		// If the cryostat is no longer cold or operational, return to the appropriate warm state.
		IF stat.nState = E_NOTT_CRYO_CTRL_STATE.COLD
		   AND NOT (stat.bOP OR stat.bCold) THEN
			ctrl.bEnable_WarmUp := FALSE;
		
			IF stat.bVacuumOK OR stat.bVacuum THEN
				logs.M_LogInfo('Cryostat no longer cold. State is WARM_VACUUM.');
				stat.nState := E_NOTT_CRYO_CTRL_STATE.WARM_VACUUM;
			ELSE
				ctrl.bEnable_CoolDown := FALSE;
				logs.M_LogInfo('Cryostat no longer cold and vacuum not present. State is WARM_PRESS.');
				stat.nState := E_NOTT_CRYO_CTRL_STATE.WARM_PRESS;
			END_IF
		
		// Process queued top-level commands.
		ELSIF stat.nState = E_NOTT_CRYO_CTRL_STATE.COLD
		   AND ctrl.bExecute THEN
			ctrl.bExecute     := FALSE;
			stat.nLastCommand := ctrl.nCommand;
			ctrl.nCommand     := E_NOTT_CRYO_CTRL_CMD.NONE;
		
			CASE stat.nLastCommand OF
		
				E_NOTT_CRYO_CTRL_CMD.WARM_UP:
					IF warm_up.bPermitStart THEN
						logs.M_LogInfo('Warm-up started.');
		
						ctrl.bEnable_Evac     := TRUE;
						ctrl.bEnable_WarmUp   := TRUE;
						ctrl.bEnable_CoolDown := FALSE;
		
						stat.nState := E_NOTT_CRYO_CTRL_STATE.WARMING_UP;
					ELSE
						ctrl.bEnable_WarmUp := FALSE;
						logs.M_LogInfo('WARM_UP command rejected: warmup start not permitted in COLD.');
					END_IF
		
				E_NOTT_CRYO_CTRL_CMD.COOL:
					// Already cold. Cooling command is only useful if cooldown is not active
					// and permissions allow it.
					IF cool_down.bPermitStart AND cool_down.cooler.stat.bInitialised THEN
						logs.M_LogInfo('Cooldown command accepted in COLD: maintaining cold state.');
		
						ctrl.bEnable_Evac     := TRUE;
						ctrl.bEnable_CoolDown := TRUE;
						ctrl.bEnable_WarmUp   := FALSE;
					ELSE
						logs.M_LogInfo('COOL command ignored/rejected: system is already COLD or cooldown not permitted.');
					END_IF
		
			ELSE
				logs.M_LogInfo('Command rejected: unsupported command in COLD.');
			END_CASE
		
		// After cooler startup has completed, clear cooldown if the cooler stops
		// unexpectedly. START_PTC inactivity is part of normal startup.
		ELSIF stat.nState = E_NOTT_CRYO_CTRL_STATE.COLD
		   AND ctrl.bEnable_CoolDown
		   AND ((cool_down.stat.nState = E_NOTT_CRYO_COOLDOWN_STATE.COOLING)
			OR (cool_down.stat.nState = E_NOTT_CRYO_COOLDOWN_STATE.OPERATIONAL_TEMPERATURE_ACHIEVED))
		   AND NOT cool_down.cooler.stat.bActive THEN
			ctrl.bEnable_CoolDown := FALSE;
			logs.M_LogInfo('Cooldown enable cleared in COLD: cooler inactive.');
		END_IF
		
		M_SetStatus(stat.nState);
		RETURN;
	
	/////////////////////////////////
	E_NOTT_CRYO_CTRL_STATE.WARMING_UP:
	/////////////////////////////////
	//
	// Warmup routine is active or expected to be active.
	// Permissions are handled centrally in M_SetCmdPermissions().
	// The warmup routine must not be considered complete automatically when the
	// warm targets are reached. It remains active until the operator stops it.
	//
	
	// Cooldown must remain disabled during warmup.
	ctrl.bEnable_CoolDown := FALSE;
	
	// Evacuation should remain enabled/available during warmup.
	ctrl.bEnable_Evac := TRUE;
	
	// Reject queued top-level sequence commands while warmup is active.
	// Stop warmup via ctrl.bEnable_WarmUp FALSE and permission logic.
	IF ctrl.bExecute THEN
		stat.nLastCommand := ctrl.nCommand;
		ctrl.bExecute     := FALSE;
		ctrl.nCommand     := E_NOTT_CRYO_CTRL_CMD.NONE;
	
		CASE stat.nLastCommand OF
			E_NOTT_CRYO_CTRL_CMD.WARM_UP:
				logs.M_LogInfo('WARM_UP command ignored: warmup already active.');
	
			E_NOTT_CRYO_CTRL_CMD.COOL:
				logs.M_LogInfo('COOL command rejected: warmup active.');
		ELSE
				logs.M_LogInfo('Command rejected: warmup active.');
		END_CASE
	END_IF
	
	// Operator stop accepted by command/permission.
	IF NOT ctrl.bEnable_WarmUp THEN
		ctrl.bEnable_CoolDown := FALSE;
	
		IF stat.bOP OR stat.bCold THEN
			// Warmup was interrupted while still cold.
			ctrl.bEnable_Evac   := TRUE;
			ctrl.bEnable_WarmUp := FALSE;
	
			logs.M_LogInfo('Warmup stopped while cryostat is still cold. State is COLD.');
			stat.nState := E_NOTT_CRYO_CTRL_STATE.COLD;
	
		ELSIF stat.bVacuumOK OR stat.bVacuum THEN
			ctrl.bEnable_WarmUp := FALSE;
	
			logs.M_LogInfo('Warmup stopped. State is WARM_VACUUM.');
			stat.nState := E_NOTT_CRYO_CTRL_STATE.WARM_VACUUM;
	
		ELSE
			ctrl.bEnable_Evac   := FALSE;
			ctrl.bEnable_WarmUp := FALSE;
	
			logs.M_LogInfo('Warmup stopped and vacuum not present. State is WARM_PRESS.');
			stat.nState := E_NOTT_CRYO_CTRL_STATE.WARM_PRESS;
		END_IF
	
	// Warmup routine reports inactive while the top-level warmup command is still
	// enabled. Do not auto-stop or reclassify here. This can happen during startup,
	// a scan-order transient, or a routine implementation detail. The operator stop
	// above is the normal exit path from WARMING_UP.
	ELSIF NOT warm_up.stat.bActive THEN
		ctrl.bEnable_WarmUp   := TRUE;
		ctrl.bEnable_CoolDown := FALSE;
		ctrl.bEnable_Evac     := TRUE;
		stat.nState           := E_NOTT_CRYO_CTRL_STATE.WARMING_UP;
	END_IF
	
	M_SetStatus(stat.nState);
	RETURN;
	
	
	/////////////////////////////////
	E_NOTT_CRYO_CTRL_STATE.ERROR:
	/////////////////////////////////
	//
	// Fault state.
	// Keep commands and process routines disabled.
	// Use RESET to restart state estimation through NONE.
	//
	
	// Clear pending top-level command.
	ctrl.bExecute := FALSE;
	ctrl.nCommand := E_NOTT_CRYO_CTRL_CMD.NONE;
	
	// Disable process enables.
	// Depending on the failure type, evacuation might eventually need special
	// handling, but for now keep this simple and conservative.
	ctrl.bEnable_CoolDown := FALSE;
	ctrl.bEnable_WarmUp   := FALSE;
	ctrl.bEnable_Evac     := FALSE;
	
	// Permissions are handled centrally in M_SetCmdPermissions().
	// If desired later, add explicit ERROR handling there to force all permits FALSE.
	
	IF ctrl.bReset THEN
		ctrl.bReset := FALSE;
	
		// Re-run startup/state estimation after reset.
		stat.bSystemStarted := FALSE;
		stat.bError         := FALSE;
		stat.nState         := E_NOTT_CRYO_CTRL_STATE.NONE;
	
		logs.M_LogInfo('ERROR reset requested. Restarting state estimation.');
	
		M_SetStatus(stat.nState);
	
	// auto-recovery.

	(*
	ELSIF NOT stat.bError THEN
		stat.bSystemStarted := FALSE;
		stat.nState := E_NOTT_CRYO_CTRL_STATE.NONE;
	
		logs.M_LogInfo('ERROR cleared. Restarting state estimation.');
	
		M_SetStatus(stat.nState);
	*)
	END_IF
	
	M_SetStatus(stat.nState);
	RETURN;

END_CASE
END_METHOD

METHOD M_UpdateThermalStatus
VAR_INPUT
END_VAR
VAR
	lrDetectorTempK:		LREAL := 9999.0;
	bDetectorTempValid:		BOOL := FALSE;
	bOPInputsValid:			BOOL := FALSE;
	bOPEntryCondition:		BOOL := FALSE;
	bOPExitCondition:		BOOL := FALSE;
END_VAR
VAR_INST
	tonOPEntry:	TON;
	tonOPExit:	TON;
	tonColdEntry:	TON;
	tonColdExit:	TON;
END_VAR
VAR CONSTANT
	tOPEntryConfirm:	TIME := T#10S;
	tOPExitConfirm:		TIME := T#5S;
	tColdConfirm:		TIME := T#5S;
END_VAR

// COLD means the authoritative detector vote is below the warm threshold.
// OP is estimated centrally from the authoritative detector and base-plate
// voters together with VAGC pressure. Timers and separate reset thresholds
// prevent sensor noise from flickering the operational status.

bDetectorTempValid := nott_voters.vote_detector.stat.bValid;

IF bDetectorTempValid THEN
	lrDetectorTempK := nott_voters.vote_detector.stat.lrTempK;
END_IF

IF stat.bCold THEN
	tonColdEntry(IN := FALSE, PT := tColdConfirm);
	tonColdExit(
		IN := NOT bDetectorTempValid
			OR NOT stat.bPressureValid
			OR NOT stat.bVacuum
			OR (lrDetectorTempK > cfg.lrTemp_Warm_Reset),
		PT := tColdConfirm);

	IF tonColdExit.Q THEN
		stat.bCold := FALSE;
		tonColdExit(IN := FALSE, PT := tColdConfirm);
	END_IF
ELSE
	tonColdExit(IN := FALSE, PT := tColdConfirm);
	tonColdEntry(
		IN := bDetectorTempValid
			AND stat.bPressureValid
			AND stat.bVacuum
			AND (lrDetectorTempK < cfg.lrTemp_Warm),
		PT := tColdConfirm);

	IF tonColdEntry.Q THEN
		stat.bCold := TRUE;
		tonColdEntry(IN := FALSE, PT := tColdConfirm);
	END_IF
END_IF

// All required measurements must be valid before entering OP. A sustained
// validity loss also removes OP after the exit confirmation time.
bOPInputsValid :=
	nott_voters.vote_detector.stat.bValid
	AND nott_voters.vote_base_plate.stat.bValid
	AND VAGC.stat.bValid;

bOPEntryCondition :=
	bOPInputsValid
	AND (nott_voters.vote_detector.stat.lrTempK <= cfg.lrTemp_DET_Target)
	AND (nott_voters.vote_base_plate.stat.lrTempK < cfg.lrTemp_BasePlate_OP)
	AND (VAGC.stat.lrPressure < cfg.lrPress_OP);

bOPExitCondition :=
	NOT bOPInputsValid
	OR (nott_voters.vote_detector.stat.lrTempK > cfg.lrTemp_DET_OP_Reset)
	OR (nott_voters.vote_base_plate.stat.lrTempK > cfg.lrTemp_BasePlate_OP_Reset)
	OR (VAGC.stat.lrPressure > cfg.lrPress_OP_Reset);

IF stat.bOP THEN
	tonOPEntry(IN := FALSE, PT := tOPEntryConfirm);
	tonOPExit(IN := bOPExitCondition, PT := tOPExitConfirm);

	IF tonOPExit.Q THEN
		stat.bOP := FALSE;
		tonOPExit(IN := FALSE, PT := tOPExitConfirm);
	END_IF
ELSE
	tonOPExit(IN := FALSE, PT := tOPExitConfirm);
	tonOPEntry(IN := bOPEntryCondition, PT := tOPEntryConfirm);

	IF tonOPEntry.Q THEN
		stat.bOP := TRUE;
		tonOPEntry(IN := FALSE, PT := tOPEntryConfirm);
	END_IF
END_IF
RETURN;
END_METHOD

END_FUNCTION_BLOCK

// ---- POUs/Routines/CoolDown/FB_NOTT_CRYO_COOLDOWN.TcPOU
FUNCTION_BLOCK FB_NOTT_CRYO_COOLDOWN
VAR_INPUT
	in_bEnable:		BOOL := FALSE;	// System active while in_bEnable is TRUE
	in_Cryo_Stat:	T_NOTT_CRYO_STAT;
END_VAR
VAR_OUTPUT
	out_bPermit_Evacuation_Stop:	BOOL := FALSE;
	out_bPermit_WarmUp:				BOOL := FALSE;

END_VAR

VAR_IN_OUT
	{attribute 'OPC.UA.DA' := '0'}
	nott_temps:						FB_NOTT_TEMPERATURES;
	{attribute 'OPC.UA.DA' := '0'}
	nott_heaters:					FB_NOTT_HEATERS;
	{attribute 'OPC.UA.DA' := '0'}
	nott_t_ctrls:      				FB_NOTT_TCTRLs;
	{attribute 'OPC.UA.DA' := '0'}
	nott_t_votes: 					FB_NOTT_VOTERS;
END_VAR
VAR
	
	{attribute 'TcHmiSymbol.Show'}	
	cfg:	T_NOTT_CRYO_COOLDOWN_CFG;
	{attribute 'TcHmiSymbol.Show'}
	ctrl:	T_NOTT_CRYO_COOLDOWN_CTRL;

	{attribute 'OPC.UA.DA' := '1'}
	{attribute 'OPC.UA.DA.Access' := '1'}
	{attribute 'TcHmiSymbol.Show'}
	stat:	T_NOTT_CRYO_COOLDOWN_STAT;

// Cooler	
	
	{attribute 'TcHmiSymbol.Show'}
	cooler:			FB_METIS_CRYO_CPA;
	
//
// Internals
//
	timer:	TON;
	trig:	R_TRIG;	// Start trigger
//

	{attribute 'TcHmiSymbol.Show'}
	bPermitStart:	BOOL := FALSE;
	{attribute 'TcHmiSymbol.Show'}
	bPermitStop:	BOOL := FALSE;
	
END_VAR

M_Configure();
M_ExecuteControllers();
M_SafetyCheck();
M_StateMachine( 
	nott_temps  := nott_temps,
	nott_heaters := nott_heaters,
	nott_t_ctrls := nott_t_ctrls,
	nott_t_votes := nott_t_votes
);
M_UpdateStatus();

METHOD M_Configure
VAR_INPUT
END_VAR
VAR
	refBOOL:	REFERENCE TO BOOL;
END_VAR
// IF stat.bConfigured THEN
// 
// ELSE
// 	RETURN;
// END_IF
END_METHOD

METHOD M_ExecuteControllers
VAR
	ptrSimTemp:	POINTER TO LREAL;
END_VAR


	
// Hardware-level cooling veto. This prevents a stale command or scan-order
// delay from enabling the cooler before confirmed vacuum is available.
ctrl.cor_Cooler(
    in_bEnable := ctrl.bEnable_Cooler
        AND in_Cryo_Stat.bPressureValid
        AND in_Cryo_Stat.bVacuum
        AND (
            (in_Cryo_Stat.bIsPVPRunning
             AND in_Cryo_Stat.bIsTMPRunning)
            OR in_Cryo_Stat.bOP
        ));
Cooler(
	in_bEnable:= ctrl.cor_Cooler.out_bEnable,
	in_bSimulation:= FALSE, 
	in_sName:= 'PTC Cooler', 
	in_sSN_Compressor:= 'CPA28H5W2DNCE-410730000001', 
	in_sSN_PulseTube:= 'PT810-19880200001', 
	in_nYear_Compressor:= 2023, 
	in_nYear_PulseTube:= 2023, 
	in_lrNextService_Compressor:= 20000.0, 
	in_lrNextService_PulseTube:= 40000.0, 
	in_nSlaveID:= 16, 
	in_nPeriod:= 1000);
END_METHOD

METHOD M_PermitStart_Cooldown
VAR_INPUT
	in_bPermissionStart: BOOL;
END_VAR
bPermitStart := in_bPermissionStart;
END_METHOD

METHOD M_PermitStop_Cooldown
VAR_INPUT
	in_bPermissionStop: BOOL;
END_VAR
bPermitStop := in_bPermissionStop;
END_METHOD

METHOD M_SafetyCheck
VAR_INPUT
END_VAR
VAR CONSTANT
	lrPress_ColdAlarmTrip:	LREAL := 10.0E-1;	// [mbar]
	lrPress_ColdAlarmReset:	LREAL := 8.0E-1;	// [mbar], hysteresis reset
END_VAR
// Keep pressure and pump alarm causes separate so clearing one condition
// cannot hide the other.
IF NOT in_Cryo_Stat.bCold THEN
	stat.bPressureAlarm := FALSE;
ELSIF in_Cryo_Stat.bPressureValid THEN
	IF stat.bPressureAlarm THEN
		IF in_Cryo_Stat.lrPressure_mbar < lrPress_ColdAlarmReset THEN
			stat.bPressureAlarm := FALSE;
		END_IF
	ELSIF in_Cryo_Stat.lrPressure_mbar > lrPress_ColdAlarmTrip THEN
		stat.bPressureAlarm := TRUE;
	END_IF
END_IF

// A pump loss during active cooldown trips the routine. The alarm resets only
// after both pumps recover; a new operator command is required to restart.
IF stat.bActive
    AND NOT in_Cryo_Stat.bOP
    AND (NOT in_Cryo_Stat.bIsPVPRunning
         OR NOT in_Cryo_Stat.bIsTMPRunning) THEN

    stat.bPumpAlarm := TRUE;
    ctrl.bEnable_Cooler := FALSE;
    stat.nState := E_NOTT_CRYO_COOLDOWN_STATE.STOP_COOLDOWN;
    stat.sErrorText := 'Pump stopped during cooldown.';

ELSIF (in_Cryo_Stat.bIsPVPRunning
       AND in_Cryo_Stat.bIsTMPRunning)
      OR in_Cryo_Stat.bOP THEN

    stat.bPumpAlarm := FALSE;
END_IF


stat.bAlarm := stat.bPressureAlarm OR stat.bPumpAlarm;
stat.bWarning := stat.bAlarm;
END_METHOD

METHOD M_StateMachine : BOOL
VAR_INPUT
END_VAR
VAR_IN_OUT
	{attribute 'OPC.UA.DA' := '0'}
	nott_temps:						FB_NOTT_TEMPERATURES;
	{attribute 'OPC.UA.DA' := '0'}
	nott_heaters:					FB_NOTT_HEATERS;
	{attribute 'OPC.UA.DA' := '0'}
	nott_t_ctrls:      				FB_NOTT_TCTRLs;
	{attribute 'OPC.UA.DA' := '0'}
	nott_t_votes: 					FB_NOTT_VOTERS;
END_VAR
VAR_INST
    tonStopCooldown : TON;
END_VAR
M_StateMachine := FALSE;

// The routine cannot remain in a cooling state without confirmed vacuum.
// The actuator is already vetoed in M_ExecuteControllers(); this transition
// keeps the routine state and HMI status consistent with physical safety.
IF ((stat.nState = E_NOTT_CRYO_COOLDOWN_STATE.START_PTC)
	OR (stat.nState = E_NOTT_CRYO_COOLDOWN_STATE.START_RAMPDOWN_DETECTOR)
	OR (stat.nState = E_NOTT_CRYO_COOLDOWN_STATE.COOLING)
	OR (stat.nState = E_NOTT_CRYO_COOLDOWN_STATE.OPERATIONAL_TEMPERATURE_ACHIEVED))
	AND (NOT in_Cryo_Stat.bPressureValid OR NOT in_Cryo_Stat.bVacuum) THEN
	ctrl.bEnable_Cooler := FALSE;
	stat.nState := E_NOTT_CRYO_COOLDOWN_STATE.STOP_COOLDOWN;
	stat.sStatus := 'Stopping cooldown: vacuum lost or pressure invalid.';
END_IF

CASE stat.nState OF

    E_NOTT_CRYO_COOLDOWN_STATE.NONE:
        // Nothing to do here
        stat.sStatus := 'NONE';
		stat.bActive := FALSE;
		stat.nState := E_NOTT_CRYO_COOLDOWN_STATE.OFF;

    E_NOTT_CRYO_COOLDOWN_STATE.OFF:

        ctrl.cor_Cooler.M_SetPermissions(FALSE, TRUE); // Only OFF allowed

        stat.sState  := 'OFF';
        stat.sStatus := 'OFF';

        ctrl.bEnable_Cooler := FALSE;

        out_bPermit_Evacuation_Stop := TRUE;
        out_bPermit_WarmUp          := TRUE;
		stat.bActive := FALSE;
		
        trig(CLK := in_bEnable);

        IF trig.Q
		   AND in_Cryo_Stat.bPressureValid
		   AND in_Cryo_Stat.bVacuum
		   AND in_Cryo_Stat.bIsPVPRunning
		   AND in_Cryo_Stat.bIsTMPRunning THEN
            stat.nState := E_NOTT_CRYO_COOLDOWN_STATE.START_PTC;
            stat.sStatus := 'Starting PTC...';

            out_bPermit_Evacuation_Stop := FALSE;
            out_bPermit_WarmUp          := FALSE;
			
			stat.bActive := TRUE;
		ELSIF trig.Q THEN
			stat.sStatus := 'Cooldown start rejected: vacuum/pumps not ready.';
        END_IF;


    E_NOTT_CRYO_COOLDOWN_STATE.START_PTC:
		stat.bActive := TRUE;
		ctrl.cor_Cooler.M_SetPermissions(TRUE, TRUE);

		out_bPermit_Evacuation_Stop := FALSE;
		out_bPermit_WarmUp          := FALSE;

		IF NOT in_bEnable THEN
			ctrl.bEnable_Cooler := FALSE;
			stat.nState := E_NOTT_CRYO_COOLDOWN_STATE.STOP_COOLDOWN;
			stat.sStatus := 'Cooldown cancelled while starting PTC...';
		ELSE
			ctrl.bEnable_Cooler := TRUE;

			IF cooler.stat.bSystemOn THEN
				stat.nState := E_NOTT_CRYO_COOLDOWN_STATE.START_RAMPDOWN_DETECTOR;
				stat.sStatus := 'PTC started. Starting detector ramp down...';
			END_IF
		END_IF


    E_NOTT_CRYO_COOLDOWN_STATE.START_RAMPDOWN_DETECTOR:
		ctrl.cor_Cooler.M_SetPermissions(TRUE, TRUE);
		ctrl.bEnable_Cooler := TRUE;

		IF NOT in_bEnable THEN
			ctrl.bEnable_Cooler := FALSE;
			stat.nState := E_NOTT_CRYO_COOLDOWN_STATE.STOP_COOLDOWN;
			stat.sStatus := 'Stopping cooldown...';
			RETURN;
		END_IF

        // Enable detector heaters
        nott_heaters.h_detector.M_SetEnable();
        nott_heaters.h_detector_spare.M_SetEnable();

        // Enable detector temperature control loops
        nott_t_ctrls.tc_detector.M_SetEnable();
        nott_t_ctrls.tc_detector_spare.M_SetEnable();

        // Set detector setpoints
        nott_t_ctrls.tc_detector.M_Set_SetPoint(
            m_eSetpointType    := E_METIS_CTRL_SETPOINT_SWITCH.FIXED,
            m_lrFixedSetpoint  := cfg.lrTemp_Det,
            m_lrSetpointOffset := 0.0,
            m_pSetpointTemp    := nott_temps.M_SetTemperatureSensor(0)
        );

        nott_t_ctrls.tc_detector_spare.M_Set_SetPoint(
            m_eSetpointType    := E_METIS_CTRL_SETPOINT_SWITCH.FIXED,
            m_lrFixedSetpoint  := cfg.lrTemp_Det,
            m_lrSetpointOffset := 0.0,
            m_pSetpointTemp    := nott_temps.M_SetTemperatureSensor(0)
        );

        stat.sStatus := 'Detector ramp down active...';

        stat.nState := E_NOTT_CRYO_COOLDOWN_STATE.COOLING;
		stat.bActive := TRUE;

    E_NOTT_CRYO_COOLDOWN_STATE.COOLING:
		ctrl.cor_Cooler.M_SetPermissions(TRUE, TRUE);
		ctrl.bEnable_Cooler := TRUE;

        out_bPermit_Evacuation_Stop := FALSE;
        out_bPermit_WarmUp          := FALSE;
		stat.bActive := TRUE;
        IF in_bEnable THEN

            IF in_Cryo_Stat.bOP THEN

                stat.sStatus := 'Operational temperature achieved.';
                stat.nState  := E_NOTT_CRYO_COOLDOWN_STATE.OPERATIONAL_TEMPERATURE_ACHIEVED;

            ELSE
                stat.sStatus := 'Cooling...';
            END_IF;

        ELSE
            stat.nState := E_NOTT_CRYO_COOLDOWN_STATE.STOP_COOLDOWN;
            stat.sStatus := 'Stopping cooldown...';
        END_IF;


    E_NOTT_CRYO_COOLDOWN_STATE.OPERATIONAL_TEMPERATURE_ACHIEVED:
		stat.bActive := TRUE;
		ctrl.cor_Cooler.M_SetPermissions(TRUE, TRUE);
		ctrl.bEnable_Cooler := TRUE;
        IF in_bEnable THEN
			IF NOT in_Cryo_Stat.bOP THEN
				out_bPermit_Evacuation_Stop := FALSE;
				out_bPermit_WarmUp          := FALSE;
				stat.nState := E_NOTT_CRYO_COOLDOWN_STATE.COOLING;
				stat.sStatus := 'Operational state lost. Resuming cooldown...';
			ELSE
                stat.sStatus := 'Operational temperature achieved.';

                out_bPermit_Evacuation_Stop := TRUE;
                out_bPermit_WarmUp          := FALSE;
			END_IF

        ELSE
            stat.nState := E_NOTT_CRYO_COOLDOWN_STATE.STOP_COOLDOWN;
            stat.sStatus := 'Stopping cooldown...';

            out_bPermit_Evacuation_Stop := FALSE;
            out_bPermit_WarmUp          := FALSE;
        END_IF;


    E_NOTT_CRYO_COOLDOWN_STATE.STOP_COOLDOWN:
		stat.bActive := TRUE;
		// Disable PTC
		ctrl.cor_Cooler.M_SetPermissions(FALSE, TRUE);
		ctrl.bEnable_Cooler := FALSE;
	
		out_bPermit_Evacuation_Stop := FALSE;
		out_bPermit_WarmUp          := FALSE;
	
		// Keep detector protection active
		nott_heaters.h_detector.M_SetEnable();
		nott_heaters.h_detector_spare.M_SetEnable();
	
		nott_t_ctrls.tc_detector.M_SetEnable();
		nott_t_ctrls.tc_detector_spare.M_SetEnable();
	
		// Follow the lowest cryostat temperature +10 K
		nott_t_ctrls.tc_detector.M_Set_SetPoint(
			m_eSetpointType    := E_METIS_CTRL_SETPOINT_SWITCH.FIXED,
			m_lrFixedSetpoint  := nott_temps.out_lrLowestTemp,
			m_lrSetpointOffset := 10.0,
			m_pSetpointTemp    := nott_temps.M_SetTemperatureSensor(0));
	
		nott_t_ctrls.tc_detector_spare.M_Set_SetPoint(
			m_eSetpointType    := E_METIS_CTRL_SETPOINT_SWITCH.FIXED,
			m_lrFixedSetpoint  := nott_temps.out_lrLowestTemp,
			m_lrSetpointOffset := 10.0,
			m_pSetpointTemp    := nott_temps.M_SetTemperatureSensor(0));
	
		stat.sStatus := 'Waiting for detector protection...';
	
		// Safety timeout (e.g. 5 minutes)
		tonStopCooldown(IN := TRUE, PT := T#15M);
	
		IF ((nott_t_votes.vote_detector.stat.bValid
			AND nott_temps.out_bLowestTempValid
			AND (nott_t_votes.vote_detector.stat.lrTempK >= (nott_temps.out_lrLowestTemp + 8.0)))
			OR tonStopCooldown.Q) THEN
	
			tonStopCooldown(IN := FALSE);
	
			stat.sStatus := 'Cooldown stopped.';
			stat.nState := E_NOTT_CRYO_COOLDOWN_STATE.OFF;
			stat.bActive := FALSE;
		END_IF;


ELSE
    stat.nState  := E_NOTT_CRYO_COOLDOWN_STATE.NONE;
    stat.sStatus := 'UNKNOWN STATE';
	stat.bActive := FALSE;
END_CASE;

M_StateMachine := TRUE;
END_METHOD

METHOD M_UpdateStatus : BOOL
VAR_INPUT
END_VAR
stat.bEnabled		:= in_bEnable;
END_METHOD

END_FUNCTION_BLOCK

// ---- POUs/Devices/Temperatures/FB_NOTT_TEMPERATURES.TcPOU
FUNCTION_BLOCK FB_NOTT_TEMPERATURES
VAR_OUTPUT
	{attribute 'OPC.UA.DA' := '0'}
	out_lrHighestTemp:		LREAL;
	out_sHighestTempName:	STRING;
	out_bHighestTempValid:	BOOL;
	
	{attribute 'OPC.UA.DA' := '0'}
	out_lrLowestTemp:		LREAL;
	out_sLowestTempName:	STRING;
	out_bLowestTempValid:	BOOL;
	
	out_lrAverageOfAllTemps: LREAL;
	
	out_all_temperature_names   : ARRAY [0..30] OF STRING;
END_VAR
VAR
	
	{attribute 'OPC.UA.DA' := '0'}
	{attribute 'TcHmiSymbol.Show'}
	all_temperatures		: ARRAY [MIN_INDEX..MAX_INDEX] OF POINTER TO FB_METIS_TEMPERATURE;
    
    // NOTE: the names below are needed for the VISU, which cannot deal with MIN_INDEX and MAX_INDEX
    // Hence, we must specify the numbers explicitly
    // MAKE SURE THE INDEXES ALWATS CORRESPOND TO THE CONSTANTS MIN_INDEX AND MAX_INDEX
	{attribute 'OPC.UA.DA' := '0'}
	{attribute 'TcHmiSymbol.Show'}
    all_temperature_names   : ARRAY [0..30] OF STRING;  // names of the temperatures

(* Empty temp: 1 *)
    
{attribute 'OPC.UA.DA' := '0'}
{attribute 'TcHmiSymbol.Show'}
empty_temp					: FB_METIS_TEMPERATURE;

//
// PT100 Temperatures
//
		
	// SideCar (* 3 *)
	{attribute 'OPC.UA.DA' := '1'}
	{attribute 'TcHmiSymbol.Show'}
	t_sidecar_1:			FB_METIS_TEMPERATURE;
	{attribute 'OPC.UA.DA' := '1'}
	{attribute 'TcHmiSymbol.Show'}
	t_sidecar_2:			FB_METIS_TEMPERATURE;
	{attribute 'OPC.UA.DA' := '1'}
	{attribute 'TcHmiSymbol.Show'}
	t_sidecar_vote:			FB_METIS_TEMPERATURE;
	
	// Photonic Chip (* 3 *)
	{attribute 'OPC.UA.DA' := '1'}
	{attribute 'TcHmiSymbol.Show'}
	t_photonic_chip_1:			FB_METIS_TEMPERATURE;
	{attribute 'OPC.UA.DA' := '1'}
	{attribute 'TcHmiSymbol.Show'}
	t_photonic_chip_2:			FB_METIS_TEMPERATURE;
	{attribute 'OPC.UA.DA' := '1'}
	{attribute 'TcHmiSymbol.Show'}
	t_photonic_chip_vote:		FB_METIS_TEMPERATURE;	
	
	// Base Plate (* 3 *)
	{attribute 'OPC.UA.DA' := '1'}
	{attribute 'TcHmiSymbol.Show'}
	t_base_plate_1:			FB_METIS_TEMPERATURE;
	{attribute 'OPC.UA.DA' := '1'}
	{attribute 'TcHmiSymbol.Show'}
	t_base_plate_2:			FB_METIS_TEMPERATURE;
	{attribute 'OPC.UA.DA' := '1'}
	{attribute 'TcHmiSymbol.Show'}
	t_base_plate_vote:			FB_METIS_TEMPERATURE;
	
	// Shield (* 3 *)
	{attribute 'OPC.UA.DA' := '1'}
	{attribute 'TcHmiSymbol.Show'}
	t_shield_1:			FB_METIS_TEMPERATURE;
	{attribute 'OPC.UA.DA' := '1'}
	{attribute 'TcHmiSymbol.Show'}
	t_shield_2:			FB_METIS_TEMPERATURE;
	{attribute 'OPC.UA.DA' := '1'}
	{attribute 'TcHmiSymbol.Show'}
	t_shield_vote:			FB_METIS_TEMPERATURE;
	
//
// DT670 Temperature sensors connected via LS240-2P
//
		// Detector (* 3 *)
	{attribute 'OPC.UA.DA' := '1'}
	{attribute 'TcHmiSymbol.Show'}
	t_detector:					FB_METIS_TEMPERATURE;
	{attribute 'OPC.UA.DA' := '1'}
	{attribute 'TcHmiSymbol.Show'}
	t_detector_spare:			FB_METIS_TEMPERATURE;
	{attribute 'OPC.UA.DA' := '1'}
	{attribute 'TcHmiSymbol.Show'}
	t_detector_vote:		FB_METIS_TEMPERATURE;

	// System temperatures   (* 3 *)
	// Legacy system-temperature channels; not used for cryostat state estimation.
	{attribute 'OPC.UA.DA' := '1'}
	{attribute 'TcHmiSymbol.Show'}
	t_master                 	:FB_METIS_TEMPERATURE;
	{attribute 'OPC.UA.DA' := '1'}
	{attribute 'TcHmiSymbol.Show'}
	t_master_vot_1           	:FB_METIS_TEMPERATURE;
	{attribute 'OPC.UA.DA' := '1'}
	{attribute 'TcHmiSymbol.Show'}
	t_master_vot_2           	:FB_METIS_TEMPERATURE;
	
	// Flat Field   (* 3 *)
	{attribute 'OPC.UA.DA' := '1'}
	{attribute 'TcHmiSymbol.Show'}
	t_flat_field_1:			FB_METIS_TEMPERATURE;
	{attribute 'OPC.UA.DA' := '1'}
	{attribute 'TcHmiSymbol.Show'}
	t_flat_field_2:			FB_METIS_TEMPERATURE;
	{attribute 'OPC.UA.DA' := '1'}
	{attribute 'TcHmiSymbol.Show'}
	t_flat_field_vote:			FB_METIS_TEMPERATURE;
	
	// Thermal Box   (* 5 *)
	{attribute 'OPC.UA.DA' := '1'}
	{attribute 'TcHmiSymbol.Show'}
	t_thermal_box_1:			FB_METIS_TEMPERATURE;
	{attribute 'OPC.UA.DA' := '1'}
	{attribute 'TcHmiSymbol.Show'}
	t_thermal_box_2:			FB_METIS_TEMPERATURE;
	{attribute 'OPC.UA.DA' := '1'}
	{attribute 'TcHmiSymbol.Show'}
	t_thermal_box_3:			FB_METIS_TEMPERATURE;
	{attribute 'OPC.UA.DA' := '1'}
	{attribute 'TcHmiSymbol.Show'}
	t_thermal_box_4:			FB_METIS_TEMPERATURE;
	{attribute 'OPC.UA.DA' := '1'}
	{attribute 'TcHmiSymbol.Show'}
	t_thermal_box_vote:			FB_METIS_TEMPERATURE;
	
		// Cabinet   (* 3 *)
	{attribute 'OPC.UA.DA' := '1'}	
	{attribute 'TcHmiSymbol.Show'}
	t_cabinet_1:			FB_METIS_TEMPERATURE;
	{attribute 'OPC.UA.DA' := '1'}
	{attribute 'TcHmiSymbol.Show'}
	t_cabinet_2:			FB_METIS_TEMPERATURE;
	{attribute 'OPC.UA.DA' := '1'}
	{attribute 'TcHmiSymbol.Show'}
	t_cabinet_vote:			FB_METIS_TEMPERATURE;

(*Vars*)

{attribute 'OPC.UA.DA' := '0'}
bConfigured					: BOOL := FALSE;

               
END_VAR
VAR CONSTANT
	{attribute 'OPC.UA.DA' := '0'}
    MIN_INDEX : INT := 0;
	{attribute 'OPC.UA.DA' := '0'}
    MAX_INDEX : INT := 30; // 1 + 3 + 3 + 3 + 3 + 3 + 3 + 3 + 5 + 3 = 30 items ==> MAX_INDEX = 30
END_VAR

M_Configure();

// to avoid invalid pointers, it is recommended to update the pointers every cycle
M_UpdatePointers();

M_ReadSensors();

M_MaxMinAvrgTemperatures();


//sim_t_cry_sha_1(in_Temp_Sensor_DT670 := t_cry_sha_1);
//sim_t_cry_sha_2(in_Temp_Sensor_DT670 := t_cry_sha_2);
//sim_t_sca_fw_icar(in_Temp_Sensor_DT670 := t_sca_fw_icar);
//sim_t_img_n_pw_icar(in_Temp_Sensor_DT670 := t_img_n_pw_icar);
//sim_t_lms_pla_1(in_Temp_Sensor_DT670 := t_lms_pla_1);

METHOD M_ConfigSimTemperatures
VAR_INPUT
END_VAR


//sim_t_cry_sha_1(in_Temp_Sensor_DT670 := t_cry_sha_1);
//sim_t_cry_sha_2(in_Temp_Sensor_DT670 := t_cry_sha_2);
//sim_t_sca_fw_icar(in_Temp_Sensor_DT670 := t_sca_fw_icar);
//sim_t_img_n_pw_icar(in_Temp_Sensor_DT670 := t_img_n_pw_icar);
//sim_t_lms_pla_1(in_Temp_Sensor_DT670 := t_lms_pla_1);
END_METHOD

METHOD M_Configure : BOOL
VAR_INPUT
END_VAR
VAR
    i : INT;
END_VAR
IF NOT bConfigured THEN
    
    // just as a safety precaution, set valid pointers to start with
    FOR i := MIN_INDEX TO MAX_INDEX DO
        all_temperatures[i] := ADR(empty_temp);
    END_FOR
    
    // Configure the all temp array
    M_UpdatePointers();
    
    // execute the M_ReadSensors function once to update the names
    M_ReadSensors();
    
    // store the names in a separate array
    FOR i := MIN_INDEX TO MAX_INDEX DO
        all_temperature_names[i] := all_temperatures[i]^.in_sName;
    END_FOR

    // Config SIM Temperatures
    M_ConfigSimTemperatures();
    
    bConfigured := TRUE;
END_IF
END_METHOD

METHOD M_GetTempSensorIndex : INT
VAR_INPUT
    sName : STRING;
END_VAR
VAR
    i: INT;
END_VAR
FOR i := MIN_INDEX TO MAX_INDEX DO
    IF sName = all_temperatures[i]^.in_sName THEN
        M_GetTempSensorIndex := i;
        RETURN;
    END_IF
END_FOR

// Handle error: sensor name not found
M_GetTempSensorIndex := 0; // empty temperature
END_METHOD

METHOD M_IsIgnoredTemperature : BOOL
VAR_INPUT
    index : INT;   // Index into all_temperatures[]
END_VAR
VAR

    IgnoreList: 		ARRAY[1..11] OF STRING := [
	   't_thermal_box_1', 	
	   't_thermal_box_2', 	
	   't_thermal_box_3', 	
	   't_thermal_box_4', 	
	   't_thermal_box_vote',  
	   't_master',
	   't_master_vot_1',
	   't_master_vot_2',
	   
	   't_cabinet_1', 	
	   't_cabinet_2', 	
	   't_cabinet_vote'   	   
	   
    ];
    i : INT;
END_VAR
M_IsIgnoredTemperature := FALSE;

// Loop through ignore list
FOR i := 1 TO 11 DO
    IF all_temperatures[index]^.in_sName = IgnoreList[i] THEN
        M_IsIgnoredTemperature := TRUE;
        RETURN; // Exit early once a match is found
    END_IF
END_FOR
END_METHOD

METHOD M_MaxMinAvrgTemperatures
VAR_INPUT
END_VAR
VAR
	lrHigestTemp:		LREAL;	// Temporary var Higest temp
	sHighestTempName:	STRING;
	
	lrLowestTemp:		LREAL;	// Temporary var Lowest temp
	sLowestTempName:	STRING;
	
	lrAverageTemp:		LREAL;	// Temporary var Lowest temp
	nSample:	INT;	// Number of valid sensor readings
	i:			INT;
	
	
END_VAR
(*Highest Temperature*)

lrHigestTemp	:= -10000.0; // setting initial temperature for comparision
sHighestTempName := '';
lrLowestTemp := 10000.0; // setting initial temperature for comparision
sLowestTempName := '';
lrAverageTemp:= 0.0; 	// setting initial temperature for comparision		

nSample	:= 0;

FOR i := MIN_INDEX TO MAX_INDEX DO
		// Ignor Ambient temps
		IF M_IsIgnoredTemperature(index := i) THEN		
			; // Skip this sensor in averaging, highest, lowest calculation
		ELSE			
			IF  all_temperatures[i]^.stat.bValid	THEN
				
					IF  all_temperatures[i]^.stat.lrTempK > lrHigestTemp THEN
						lrHigestTemp	:= all_temperatures[i]^.stat.lrTempK;
						sHighestTempName := all_temperatures[i]^.in_sName;
					END_IF
					
					IF  all_temperatures[i]^.stat.lrTempK < lrLowestTemp THEN
						lrLowestTemp	:= all_temperatures[i]^.stat.lrTempK;
						sLowestTempName    := all_temperatures[i]^.in_sName;
					END_IF
					
					lrAverageTemp	:= lrAverageTemp + all_temperatures[i]^.stat.lrTempK;	
					
					nSample	:= nSample + 1;
			END_IF
			
		END_IF
END_FOR



IF nSample > 0	THEN
	out_lrAverageOfAllTemps	:= lrAverageTemp / nSample;
	
	out_lrHighestTemp := lrHigestTemp;		
	out_sHighestTempName := sHighestTempName;
	out_bHighestTempValid := TRUE;
	
	out_lrLowestTemp :=		lrLowestTemp;
	out_sLowestTempName :=	sLowestTempName;
	out_bLowestTempValid := TRUE;
	
	
	
ELSE
	
	out_lrAverageOfAllTemps	:= 9999;
	
	out_lrHighestTemp := 9999;		
	out_sHighestTempName := 'NA';
	out_bHighestTempValid := FALSE;
	
	out_lrLowestTemp :=		9999;
	out_sLowestTempName :=	'NA';
	out_bLowestTempValid := FALSE;
END_IF
END_METHOD

METHOD M_ReadSensors
VAR_INPUT
END_VAR
empty_temp			(in_sName:='', in_eType := E_METIS_SENSOR_TYPE.TEMPERATURE, in_eSource := E_METIS_SENSOR_SOURCE.LS240, in_nRampPeriodSec:= 10, in_lrFaultRamp:= 10);
	// SideCar (* 3 *)	
t_sidecar_1           (in_sName:='t_sidecar_1', 	in_eType := E_METIS_SENSOR_TYPE.TEMPERATURE, in_eSource := E_METIS_SENSOR_SOURCE.EL32XX, in_lrScale := 0.01, in_lrOffset := 273.15);
t_sidecar_2           (in_sName:='t_sidecar_2', 	in_eType := E_METIS_SENSOR_TYPE.TEMPERATURE, in_eSource := E_METIS_SENSOR_SOURCE.EL32XX, in_lrScale := 0.01, in_lrOffset := 273.15);
t_sidecar_vote        (in_sName:='t_sidecar_vote',  in_eType := E_METIS_SENSOR_TYPE.TEMPERATURE, in_eSource := E_METIS_SENSOR_SOURCE.VOTER,  in_nRampPeriodSec:= 10, in_lrFaultRamp:= 10);

	// Photonic Chip (* 3 *)
t_photonic_chip_1           (in_sName:='t_photonic_chip_1', 	in_eType := E_METIS_SENSOR_TYPE.TEMPERATURE, in_eSource := E_METIS_SENSOR_SOURCE.EL32XX, in_lrScale := 0.01, in_lrOffset := 273.15);
t_photonic_chip_2           (in_sName:='t_photonic_chip_2', 	in_eType := E_METIS_SENSOR_TYPE.TEMPERATURE, in_eSource := E_METIS_SENSOR_SOURCE.EL32XX, in_lrScale := 0.01, in_lrOffset := 273.15);
t_photonic_chip_vote        (in_sName:='t_photonic_chip_vote',  	in_eType := E_METIS_SENSOR_TYPE.TEMPERATURE, in_eSource := E_METIS_SENSOR_SOURCE.VOTER,  in_nRampPeriodSec:= 10, in_lrFaultRamp:= 10);

	// Base Plate (* 3 *)
t_base_plate_1           (in_sName:='t_base_plate_1', 	in_eType := E_METIS_SENSOR_TYPE.TEMPERATURE, in_eSource := E_METIS_SENSOR_SOURCE.EL32XX, in_lrScale := 0.01, in_lrOffset := 273.15);
t_base_plate_2           (in_sName:='t_base_plate_2', 	in_eType := E_METIS_SENSOR_TYPE.TEMPERATURE, in_eSource := E_METIS_SENSOR_SOURCE.EL32XX, in_lrScale := 0.01, in_lrOffset := 273.15);
t_base_plate_vote        (in_sName:='t_base_plate_vote',  	in_eType := E_METIS_SENSOR_TYPE.TEMPERATURE, in_eSource := E_METIS_SENSOR_SOURCE.VOTER,  in_nRampPeriodSec:= 10, in_lrFaultRamp:= 10);

	// Shield (* 3 *)
t_shield_1           (in_sName:='t_shield_1', 	in_eType := E_METIS_SENSOR_TYPE.TEMPERATURE, in_eSource := E_METIS_SENSOR_SOURCE.EL32XX, in_lrScale := 0.01, in_lrOffset := 273.15);
t_shield_2           (in_sName:='t_shield_2', 	in_eType := E_METIS_SENSOR_TYPE.TEMPERATURE, in_eSource := E_METIS_SENSOR_SOURCE.EL32XX, in_lrScale := 0.01, in_lrOffset := 273.15);
t_shield_vote        (in_sName:='t_shield_vote',  	in_eType := E_METIS_SENSOR_TYPE.TEMPERATURE, in_eSource := E_METIS_SENSOR_SOURCE.VOTER,  in_nRampPeriodSec:= 10, in_lrFaultRamp:= 10);

//
// DT670 Temperature sensors connected via LS240-2P
//
		// Detector (* 3 *)
t_detector			(in_sName:='t_detector', in_eType := E_METIS_SENSOR_TYPE.TEMPERATURE, in_eSource := E_METIS_SENSOR_SOURCE.LS240, in_nRampPeriodSec:= 10, in_lrFaultRamp:= 10);
t_detector_spare	(in_sName:='t_detector_spare', in_eType := E_METIS_SENSOR_TYPE.TEMPERATURE, in_eSource := E_METIS_SENSOR_SOURCE.LS240, in_nRampPeriodSec:= 10, in_lrFaultRamp:= 10);			
t_detector_vote     (in_sName:='t_detector_vote',  in_eType := E_METIS_SENSOR_TYPE.TEMPERATURE, in_eSource := E_METIS_SENSOR_SOURCE.VOTER, in_nRampPeriodSec:= 10, in_lrFaultRamp:= 10);

// System temperatures   (* 3 *)
// Legacy system-temperature channels; not used for cryostat state estimation.

t_master       		(in_sName:='t_master',  in_eType := E_METIS_SENSOR_TYPE.TEMPERATURE, in_eSource := E_METIS_SENSOR_SOURCE.VOTER, in_nRampPeriodSec:= 10, in_lrFaultRamp:= 10);
t_master_vot_1 		(in_sName:='t_master_vot_1',  in_eType := E_METIS_SENSOR_TYPE.TEMPERATURE, in_eSource := E_METIS_SENSOR_SOURCE.VOTER, in_nRampPeriodSec:= 10, in_lrFaultRamp:= 10);
t_master_vot_2 		(in_sName:='t_master_vot_2',  in_eType := E_METIS_SENSOR_TYPE.TEMPERATURE, in_eSource := E_METIS_SENSOR_SOURCE.VOTER, in_nRampPeriodSec:= 10, in_lrFaultRamp:= 10);

	// Flat Field 
	
t_flat_field_1           (in_sName:='t_flat_field_1', 	in_eType := E_METIS_SENSOR_TYPE.TEMPERATURE, in_eSource := E_METIS_SENSOR_SOURCE.EL32XX, in_lrScale := 0.01, in_lrOffset := 273.15);
t_flat_field_2           (in_sName:='t_flat_field_2', 	in_eType := E_METIS_SENSOR_TYPE.TEMPERATURE, in_eSource := E_METIS_SENSOR_SOURCE.EL32XX, in_lrScale := 0.01, in_lrOffset := 273.15);
t_flat_field_vote        (in_sName:='t_flat_field_vote',  	in_eType := E_METIS_SENSOR_TYPE.TEMPERATURE, in_eSource := E_METIS_SENSOR_SOURCE.VOTER,  in_nRampPeriodSec:= 10, in_lrFaultRamp:= 10);

// Thermal Box   (* 5 *)
t_thermal_box_1           (in_sName:='t_thermal_box_1', 	in_eType := E_METIS_SENSOR_TYPE.TEMPERATURE, in_eSource := E_METIS_SENSOR_SOURCE.EL32XX, in_lrScale := 0.01, in_lrOffset := 273.15);
t_thermal_box_2           (in_sName:='t_thermal_box_2', 	in_eType := E_METIS_SENSOR_TYPE.TEMPERATURE, in_eSource := E_METIS_SENSOR_SOURCE.EL32XX, in_lrScale := 0.01, in_lrOffset := 273.15);
t_thermal_box_3           (in_sName:='t_thermal_box_3', 	in_eType := E_METIS_SENSOR_TYPE.TEMPERATURE, in_eSource := E_METIS_SENSOR_SOURCE.EL32XX, in_lrScale := 0.01, in_lrOffset := 273.15);
t_thermal_box_4           (in_sName:='t_thermal_box_4', 	in_eType := E_METIS_SENSOR_TYPE.TEMPERATURE, in_eSource := E_METIS_SENSOR_SOURCE.EL32XX, in_lrScale := 0.01, in_lrOffset := 273.15);
t_thermal_box_vote        (in_sName:='t_thermal_box_vote',  	in_eType := E_METIS_SENSOR_TYPE.TEMPERATURE, in_eSource := E_METIS_SENSOR_SOURCE.VOTER,  in_nRampPeriodSec:= 10, in_lrFaultRamp:= 10);

// Cabinet   (* 3 *)
		
t_cabinet_1           (in_sName:='t_cabinet_1', 	in_eType := E_METIS_SENSOR_TYPE.TEMPERATURE, in_eSource := E_METIS_SENSOR_SOURCE.EL32XX, in_lrScale := 0.01, in_lrOffset := 273.15);
t_cabinet_2           (in_sName:='t_cabinet_2', 	in_eType := E_METIS_SENSOR_TYPE.TEMPERATURE, in_eSource := E_METIS_SENSOR_SOURCE.EL32XX, in_lrScale := 0.01, in_lrOffset := 273.15);
t_cabinet_vote        (in_sName:='t_cabinet_vote',  in_eType := E_METIS_SENSOR_TYPE.TEMPERATURE, in_eSource := E_METIS_SENSOR_SOURCE.VOTER,  in_nRampPeriodSec:= 10, in_lrFaultRamp:= 10);
END_METHOD

METHOD M_SetTemperatureSensor : POINTER TO FB_METIS_TEMPERATURE
VAR_INPUT
	m_nIndex	:	INT;
END_VAR
// always return a valid pointer!
IF (m_nIndex >= MIN_INDEX) AND (m_nIndex <= MAX_INDEX) THEN 
    M_SetTemperatureSensor := all_temperatures[m_nIndex];
ELSE
    M_SetTemperatureSensor := all_temperatures[0]; // empty temperature
END_IF
END_METHOD

METHOD M_UpdatePointer
VAR_INPUT
    pSensor : POINTER TO FB_METIS_TEMPERATURE;
END_VAR
VAR_IN_OUT
    i : INT;
END_VAR
IF i >= MIN_INDEX AND i <= MAX_INDEX THEN
    all_temperatures[i] := pSensor;
    i := i + 1;
END_IF
END_METHOD

METHOD M_UpdatePointers
VAR_INPUT
END_VAR
VAR_INST
    {attribute 'OPC.UA.DA' := '0'}
    i : INT := 0;
END_VAR
// EMPTY
M_UpdatePointer(i := i, pSensor := ADR(empty_temp));

	// SideCar (* 3 *)
M_UpdatePointer(i := i, pSensor := ADR(t_sidecar_1));
M_UpdatePointer(i := i, pSensor := ADR(t_sidecar_2));
M_UpdatePointer(i := i, pSensor := ADR(t_sidecar_vote));
	// Photonic Chip (* 3 *)
M_UpdatePointer(i := i, pSensor := ADR(t_photonic_chip_1));
M_UpdatePointer(i := i, pSensor := ADR(t_photonic_chip_2));
M_UpdatePointer(i := i, pSensor := ADR(t_photonic_chip_vote));
	// Base Plate (* 3 *)
M_UpdatePointer(i := i, pSensor := ADR(t_base_plate_1));
M_UpdatePointer(i := i, pSensor := ADR(t_base_plate_2));
M_UpdatePointer(i := i, pSensor := ADR(t_base_plate_vote));
	// Shield (* 3 *)
M_UpdatePointer(i := i, pSensor := ADR(t_shield_1));
M_UpdatePointer(i := i, pSensor := ADR(t_shield_2));
M_UpdatePointer(i := i, pSensor := ADR(t_shield_vote));
		// Detector (* 3 *)
M_UpdatePointer(i := i, pSensor := ADR(t_detector));
M_UpdatePointer(i := i, pSensor := ADR(t_detector_spare));
M_UpdatePointer(i := i, pSensor := ADR(t_detector_vote));

(*System temperatures   (3) *)
M_UpdatePointer(i := i, pSensor := ADR(t_master));
M_UpdatePointer(i := i, pSensor := ADR(t_master_vot_1));
M_UpdatePointer(i := i, pSensor := ADR(t_master_vot_2));
// Flat Field
M_UpdatePointer(i := i, pSensor := ADR(t_flat_field_1));
M_UpdatePointer(i := i, pSensor := ADR(t_flat_field_2));
M_UpdatePointer(i := i, pSensor := ADR(t_flat_field_vote));
// Thermal Box
M_UpdatePointer(i := i, pSensor := ADR(t_thermal_box_1));
M_UpdatePointer(i := i, pSensor := ADR(t_thermal_box_2));
M_UpdatePointer(i := i, pSensor := ADR(t_thermal_box_3));
M_UpdatePointer(i := i, pSensor := ADR(t_thermal_box_4));
M_UpdatePointer(i := i, pSensor := ADR(t_thermal_box_vote));
// Cabinet
M_UpdatePointer(i := i, pSensor := ADR(t_cabinet_1));
M_UpdatePointer(i := i, pSensor := ADR(t_cabinet_2));
M_UpdatePointer(i := i, pSensor := ADR(t_cabinet_vote));
END_METHOD

END_FUNCTION_BLOCK

// ---- POUs/Devices/Heaters/FB_NOTT_HEATERS.TcPOU
FUNCTION_BLOCK FB_NOTT_HEATERS
VAR_INPUT
END_VAR
VAR_OUTPUT
END_VAR
VAR_IN_OUT
	{attribute 'OPC.UA.DA' := '0'}
    tctrl:                  FB_NOTT_TCTRLs;
END_VAR
VAR

	
// Detector    
	{attribute 'TcHmiSymbol.Show'}
    h_detector:            	FB_METIS_HEATER;   // NOTT detector heater
	{attribute 'TcHmiSymbol.Show'}
    h_detector_spare:            FB_METIS_HEATER;   // NOTT detector heater SPARE
	
// Sidecar
	{attribute 'TcHmiSymbol.Show'}
    h_sidecar:            	FB_METIS_HEATER;  
	
// Photonic Chip
	{attribute 'TcHmiSymbol.Show'}
    h_photonic_chip:            	FB_METIS_HEATER;  

// // Flat Field
	{attribute 'TcHmiSymbol.Show'}
    h_flat_field:            	FB_METIS_HEATER; 

// Base Plate
	{attribute 'TcHmiSymbol.Show'}
    h_base_plate:            	FB_METIS_HEATER; 

// Shield
	{attribute 'TcHmiSymbol.Show'}
    h_shield:            	FB_METIS_HEATER;

  


END_VAR

M_ExecuteControllers(tctrl);

METHOD M_ExecuteControllers
VAR_INPUT
END_VAR
VAR_IN_OUT
    tctrl: FB_NOTT_TCTRLs;
END_VAR
// Detector 

h_detector(
    in_sName                := 'Detector HTR',
    in_lrHeaterResistance   := 75,
    in_lrHeaterMaxPower     := 5,
    in_eHeaterType          := E_METIS_CRYO_HEATER_TYPE.EL95X1,
    in_sAutoSetpointSource  := tctrl.tc_detector.in_sName,
    in_lrAutoSetpointValue  := tctrl.tc_detector.stat.lrControllerOut);
	
h_detector_spare(
    in_sName                := 'Detector Spare HTR',
    in_lrHeaterResistance   := 75,
    in_lrHeaterMaxPower     := 5,
    in_eHeaterType          := E_METIS_CRYO_HEATER_TYPE.EL95X1,
    in_sAutoSetpointSource  := tctrl.tc_detector_spare.in_sName,
    in_lrAutoSetpointValue  := tctrl.tc_detector_spare.stat.lrControllerOut);

// Sidecar

h_sidecar(
    in_sName                := 'Sidecar HTR',
    in_lrHeaterResistance   := 75,
    in_lrHeaterMaxPower     := 5,
    in_eHeaterType          := E_METIS_CRYO_HEATER_TYPE.EL95X1,
    in_sAutoSetpointSource  := tctrl.tc_sidecar.in_sName,
    in_lrAutoSetpointValue  := tctrl.tc_sidecar.stat.lrControllerOut);

// Photonic Chip

h_photonic_chip(
    in_sName                := 'Photonic Chip HTR',
    in_lrHeaterResistance   := 75,
    in_lrHeaterMaxPower     := 5,
    in_eHeaterType          := E_METIS_CRYO_HEATER_TYPE.EL95X1,
    in_sAutoSetpointSource  := tctrl.tc_photonic_chip.in_sName,
    in_lrAutoSetpointValue  := tctrl.tc_photonic_chip.stat.lrControllerOut);

// Base Plate

h_base_plate(
    in_sName                := 'Base Plate HTR',
    in_lrHeaterResistance   := 18.75,
    in_lrHeaterMaxPower     := 192,
    in_eHeaterType          := E_METIS_CRYO_HEATER_TYPE.CPAU60,
    in_sAutoSetpointSource  := tctrl.tc_base_plate.in_sName,
    in_lrAutoSetpointValue  := tctrl.tc_base_plate.stat.lrControllerOut);
	
// Shield

h_shield(
    in_sName                := 'Shield HTR',
    in_lrHeaterResistance   := 18.75,
    in_lrHeaterMaxPower     := 192,
    in_eHeaterType          := E_METIS_CRYO_HEATER_TYPE.CPAU60,
    in_sAutoSetpointSource  := tctrl.tc_shields.in_sName,
    in_lrAutoSetpointValue  := tctrl.tc_shields.stat.lrControllerOut);	

// Flat Field

h_flat_field(
    in_sName                := 'Flat Field HTR',
    in_lrHeaterResistance   := 100,
    in_lrHeaterMaxPower     := 0.48,
    in_eHeaterType          := E_METIS_CRYO_HEATER_TYPE.FLAT_FIELD,
    in_sAutoSetpointSource  := tctrl.tc_flatfield.in_sName,
    in_lrAutoSetpointValue  := tctrl.tc_flatfield.stat.lrControllerOut);
END_METHOD

END_FUNCTION_BLOCK

// ---- POUs/Devices/Control/FB_NOTT_TCTRLs.TcPOU
FUNCTION_BLOCK FB_NOTT_TCTRLs
VAR_INPUT
END_VAR
VAR_OUTPUT
END_VAR
VAR_IN_OUT
	{attribute 'OPC.UA.DA' := '0'}
    temperatures:   FB_NOTT_TEMPERATURES;  // all temperatures
END_VAR
VAR

	{attribute 'TcHmiSymbol.Show'}
    tc_detector:     		FB_NOTT_CTRL_TEMPERATURE; // Detector
	{attribute 'TcHmiSymbol.Show'}
    tc_detector_spare:     	FB_NOTT_CTRL_TEMPERATURE; // Controls spare heater on Detector
    {attribute 'TcHmiSymbol.Show'}
	tc_sidecar:     		FB_NOTT_CTRL_TEMPERATURE; // Sidecar
	{attribute 'TcHmiSymbol.Show'}
    tc_photonic_chip:       FB_NOTT_CTRL_TEMPERATURE; // Photonic Chip
	{attribute 'TcHmiSymbol.Show'}
    tc_base_plate:      	FB_NOTT_CTRL_TEMPERATURE; // Base Plate
	{attribute 'TcHmiSymbol.Show'}
	tc_shields:      		FB_NOTT_CTRL_TEMPERATURE; // Shield
	{attribute 'TcHmiSymbol.Show'}
	tc_flatfield:      		FB_NOTT_CTRL_TEMPERATURE; // Flatfield

END_VAR
VAR CONSTANT
	{attribute 'OPC.UA.DA' := '0'}
    CYCLE_TIME : TIME := T#10ms;
END_VAR

// CRY
tc_detector			(in_sName := 'tc_detector' 		 , in_tCycleTime := CYCLE_TIME, temperatures := temperatures);
tc_detector_spare	(in_sName := 'tc_detector_spare' , in_tCycleTime := CYCLE_TIME, temperatures := temperatures);
tc_sidecar			(in_sName := 'tc_sidecar' 		 , in_tCycleTime := CYCLE_TIME, temperatures := temperatures);
tc_photonic_chip	(in_sName := 'tc_photonic_chip'  , in_tCycleTime := CYCLE_TIME, temperatures := temperatures);
tc_shields			(in_sName := 'tc_shields'  		 , in_tCycleTime := CYCLE_TIME, temperatures := temperatures);
tc_flatfield		(in_sName := 'tc_flatfield'  	 , in_tCycleTime := CYCLE_TIME, temperatures := temperatures);
tc_base_plate		(in_sName := 'tc_base_plate'  	 , in_tCycleTime := CYCLE_TIME, temperatures := temperatures);

END_FUNCTION_BLOCK

// ---- POUs/Devices/Control/FB_NOTT_CTRL_TEMPERATURE.TcPOU
FUNCTION_BLOCK FB_NOTT_CTRL_TEMPERATURE
VAR_INPUT
	{attribute 'OPC.UA.DA' := '0'}
	in_sName : STRING;   // name of the controller
	{attribute 'OPC.UA.DA' := '0'}
    in_tCycleTime : TIME := T#10ms;
END_VAR
VAR_IN_OUT
	{attribute 'OPC.UA.DA' := '0'}
    temperatures : FB_NOTT_TEMPERATURES;  // all temperatures
END_VAR
VAR_OUTPUT
END_VAR
VAR
    // configuration
	{attribute 'OPC.UA.DA' := '0'}
	{attribute 'TcHmiSymbol.Show'}
	fbTcConfig : FB_READ_WRITE_METIS_CTRL_DT670_CFG;
    
    // standard objects
	{attribute 'TcHmiSymbol.Show'}
    stat : T_METIS_CTRL_LOOP_STAT;
	{attribute 'TcHmiSymbol.Show'}
    ctrl : T_NOTT_CTRL_LOOP_CTRL;
	{attribute 'TcHmiSymbol.Show'}
    cfg  : T_METIS_CTRL_LOOP_CFG;
    
    
	{attribute 'OPC.UA.DA' := '0'}
		{attribute 'TcHmiSymbol.Show'}
    pInputTemp : POINTER TO FB_METIS_TEMPERATURE;
	{attribute 'OPC.UA.DA' := '0'}
		{attribute 'TcHmiSymbol.Show'}
    pSetpointTemp : POINTER TO FB_METIS_TEMPERATURE;
    
    // Beckhoff controller
	{attribute 'OPC.UA.DA' := '0'}
	{attribute 'TcHmiSymbol.Show'}
	fbCtrlPid       : FB_CTRL_PID;
	{attribute 'OPC.UA.DA' := '0'}
	{attribute 'TcHmiSymbol.Show'}
	stCtrlPidParams : ST_CTRL_PID_PARAMS;
    
	// ramp generator
	ramp: FB_METIS_CTRL_RAMP_GENERATOR;
    
    // array for setpoint selection, used by the HMI
	{attribute 'OPC.UA.DA' := '0'}
		{attribute 'TcHmiSymbol.Show'}
    aSetpointSwitchNames : ARRAY[0..1] OF STRING := [ 'Fixed', 'Variable' ]; 
	
	
				// Alarm handling
	// List of alarms to be handled by Temperature
	arrEventEntry : ARRAY [0..4] OF TcEventEntry;
	// Alarm handler FB
	fbAlarmHandler : FB_AlarmHandler;
	{attribute 'TcHmiSymbol.Show'}
	{attribute 'TcHmiSymbol.ReadOnly'}
	sInstanceName : T_MaxString;
	{attribute 'TcHmiSymbol.Show'}
	bConfirmAllAlarms : BOOL;
	{attribute 'TcHmiSymbol.Show'}
	{attribute 'TcHmiSymbol.ReadOnly'}
	sEventClassName : T_MaxString;
	
	// Logs logs
	logs:	FB_CRYO_FUNCTION_LOG;
    
END_VAR

// to avoid any problem of invalid pointers, set them right away
M_UpdateTempPointers(temperatures := temperatures);

// Read/write configuration
fbTcConfig(in_sTempCtrlName:= in_sName, Temp_Ctrl_Config:= cfg);

// configure during the first cycles
IF NOT stat.bConfigured THEN
    M_Configure(temperatures := temperatures);
    RETURN;
END_IF

// read/write the config (if needed)
M_Read_Write_Config(temperatures := temperatures);


IF stat.bStarted THEN
    M_ExecuteModes();
    M_ExecuteController();
ELSE
    M_Startup();
END_IF

M_UpdateStatus();

IF ctrl.bClearForcedManualDiag THEN
    stat.sLastForcedManualTime := '';
    stat.sLastForcedManualCause := '';
    ctrl.bClearForcedManualDiag := FALSE;
END_IF

// Handle alarms
M_UpdateAlarms();


// Setting Power to the heater
//IF bEngMode AND (NOT ctrl.bEnable) THEN
//	lrControllerOut := lrManualOut; // set manual power
//ELSE
//	lrManualOut := lrControllerOut; // Bumpless transition
//END_IF

METHOD M_ConfigReadingFinished
VAR_INPUT
    bError : BOOL;
END_VAR
VAR_IN_OUT
    temperatures : FB_NOTT_TEMPERATURES;
END_VAR
VAR
    i : INT;
END_VAR
IF bError THEN
    // ERROR! Just put the indexes to 0
    ctrl.nInputTempIndex    := 0;
    ctrl.nSetpointTempIndex := 0;
    //ctrl.lrOutMaxLimit              := 100.0;    // TODO
    //ctrl.lrOutMinLimit              := 0.0;      // TODO

ELSE
    // success!
    // update some level-based ctrl variables
    ctrl.nInputTempIndex     := temperatures.M_GetTempSensorIndex(cfg.sInputTempName);
    ctrl.nSetpointTempIndex  := temperatures.M_GetTempSensorIndex(cfg.sSetpointTempName);
    ctrl.lrFixedSetpoint     := cfg.lrFixedSetpoint;
    ctrl.lrSetpointOffset    := cfg.lrSetpointOffset;
    ctrl.lrManualOut         := cfg.lrManualOut;
    // edge-based ctrl variables are better directly updated in stat
    stat.eCtrlMode           := cfg.eStartupCtrlMode;
    //ctrl.lrOutMaxLimit := cfg.lrOutMaxLimit;    // TODO
    //ctrl.lrOutMinLimit := cfg.lrOutMinLimit;    // TODO
END_IF

M_UpdateTempPointers(temperatures := temperatures);

// clear the flag
fbTcConfig.M_ClearReadingDoneFlag();
END_METHOD

METHOD M_Configure : BOOL
VAR_INST
	{attribute 'OPC.UA.DA' := '0'}
    nConfigureState : INT;
END_VAR
VAR_IN_OUT
	{attribute 'OPC.UA.DA' := '0'}
    temperatures : FB_NOTT_TEMPERATURES;
END_VAR
VAR
    i : INT;
END_VAR
arrEventEntry[0] := Tc_Events.METISCryoPIDCtrlEventClass.InputTemperatureInvalid;
arrEventEntry[1] := Tc_Events.METISCryoPIDCtrlEventClass.VariableSetpointInvalid;
arrEventEntry[2] := Tc_Events.METISCryoPIDCtrlEventClass.ControllerForcedManual;
arrEventEntry[3] := Tc_Events.METISCryoPIDCtrlEventClass.PidBlockError;
arrEventEntry[4] := Tc_Events.METISCryoPIDCtrlEventClass.RampBlockError;


CASE nConfigureState OF
    0:  
        // configure the base PID controller
        // init parameter struct
        stCtrlPidParams.tCtrlCycleTime	:= in_tCycleTime;
        stCtrlPidParams.tTaskCycleTime	:= in_tCycleTime;
        stCtrlPidParams.fOutMaxLimit    := 100.0;
        stCtrlPidParams.fOutMinLimit    := 0.0;
        // use the name of the control loop as the default description
        cfg.sDescription                := in_sName;
        // ensure some more default settings
        cfg.bEnabled                    := FALSE;
        stat.eCtrlMode                  := E_METIS_CTRL_MODE.MANUAL; 
        // start reading the config
        fbTcConfig.M_ReadConfiguration();
        nConfigureState := 1;
    1:
        IF fbTcConfig.bReadingDoneFlag THEN
            M_ConfigReadingFinished(
                bError       := fbTcConfig.bReadError,
                temperatures := temperatures);
            
            stat.bConfigured := TRUE;
        END_IF
END_CASE
END_METHOD

METHOD M_ExecuteController
VAR_INPUT
END_VAR
VAR_INST
	{attribute 'OPC.UA.DA' := '0'}
	eCtrlMode       : E_CTRL_MODE;
    
	{attribute 'OPC.UA.DA' := '0'}
    bEnableRamp : BOOL;
    
	{attribute 'OPC.UA.DA' := '0'}
    lrActualValue : LREAL;
END_VAR

// set the raw control mode
IF NOT cfg.bEnabled THEN
    stat.lrControllerOut := 0.0;
    stat.bError := FALSE;
    stat.bWarning := FALSE;
    stat.bValid := FALSE;
    RETURN;

ELSIF stat.eCtrlMode = E_METIS_CTRL_MODE.MANUAL THEN
    eCtrlMode := E_CTRL_MODE.eCTRL_MODE_MANUAL;
    // ramp generator should not be running
    bEnableRamp := FALSE;
ELSE
    eCtrlMode := E_CTRL_MODE.eCTRL_MODE_ACTIVE;
    // ramp generator should be running
    bEnableRamp := TRUE;
END_IF

// update the internal control params
stCtrlPidParams.fKp := cfg.lrKp;
stCtrlPidParams.tTn := LREAL_TO_TIME(cfg.lrTn * 1000.0);
stCtrlPidParams.tTd := LREAL_TO_TIME(cfg.lrTd * 1000.0);
stCtrlPidParams.tTv := LREAL_TO_TIME(cfg.lrTv * 1000.0);

// update more stat values
IF ctrl.nSetpointTempIndex <> 0 THEN
    stat.lrActVariableSetpoint := pSetpointTemp^.stat.lrTempK;
ELSE
    stat.lrActVariableSetpoint := 0.0;
END_IF

// calculate the input for the ramp
IF cfg.eSetpointSwitch = E_METIS_CTRL_SETPOINT_SWITCH.FIXED THEN
    stat.lrTargetSetpoint := ctrl.lrFixedSetpoint + ctrl.lrSetpointOffset;
ELSE 
    stat.lrTargetSetpoint := stat.lrActVariableSetpoint + ctrl.lrSetpointOffset;
END_IF

// update the input
stat.lrActInput := pInputTemp^.stat.lrTempK;

(* 
Following Beckhoff ramp generator is obsolete. Keeping it here until the tests with the new ramp geneator are successful.

// execute the ramp
ramp(
    in_bEnable          := bEnableRamp,
	in_fRampSetPoint	:= stat.lrTargetSetpoint,
    in_fStartPoint      := stat.lrActInput,
 	in_fRampUp_Rate	    := cfg.lrRampUpRate,
 	in_fRampDown_Rate   := cfg.lrRampDownRate,
 	out_fRampValue      => stat.lrRampValue); *)
	
stat.lrRampValue :=
    M_GenerateRampedSetpoint(
        in_bEnable                 := bEnableRamp,
        in_bRestart                := FALSE,

        in_lrTargetSetpoint        := stat.lrTargetSetpoint,
        in_lrProcessValue          := stat.lrActInput,

        in_lrRampUpRate            := cfg.lrRampUpRate,
        in_lrRampDownRate          := cfg.lrRampDownRate,

        in_lrMaxTrackingDifference := cfg.lrMaxTrackingDifference,
        in_lrTargetChangeThreshold := cfg.lrTargetChangeThreshold,

        in_tCycleTime              := in_tCycleTime
    );


// execute the PID algorithm
fbCtrlPid(
    fSetpointValue  := stat.lrRampValue,
    fActualValue    := stat.lrActInput,
    fManSyncValue   := ctrl.lrManualOut,
    bSync           := FALSE,
    eMode           := eCtrlMode,
    bHold           := ctrl.bHold,
    stParams        := stCtrlPidParams,
    fOut            => stat.lrControllerOut,
    bARWactive      => stat.bARWactive,
    bError          => stat.bError);

stat.nErrorId := TO_INT(fbCtrlPid.eErrorId);

// Enable a smooth transition from AUTO to MANUAL mode if needed
IF stat.eCtrlMode = E_METIS_CTRL_MODE.AUTO AND cfg.bSyncManualOut THEN
    ctrl.lrManualOut := stat.lrControllerOut;
END_IF
END_METHOD

METHOD M_ExecuteModes
VAR_INPUT
END_VAR
VAR_INST
    {attribute 'OPC.UA.DA' := '0'}
    fbInputTimer    : TON;
    {attribute 'OPC.UA.DA' := '0'}
    fbSetpointTimer : TON;
    {attribute 'OPC.UA.DA' := '0'}
    fbGetSystemTime : GETSYSTEMTIME;
    {attribute 'OPC.UA.DA' := '0'}
    fileTime        : T_FILETIME;
END_VAR
If stat.eCtrlMode = E_METIS_CTRL_MODE.NONE THEN
    // typical behavior when e.g. a config file did not contain a valid entry
    // To avoid problems, force MANUAL in this case
    stat.eCtrlMode := E_METIS_CTRL_MODE.MANUAL;
END_IF

// check which mode switches are accepted
// (currently very simple, but can be made more complex if needed)
stat.bAcceptCtrlMode_Auto := stat.eCtrlMode = E_METIS_CTRL_MODE.MANUAL
                             AND NOT stat.bError;
stat.bAcceptCtrlMode_Manual := stat.eCtrlMode = E_METIS_CTRL_MODE.AUTO ;

// switch to AUTO / MANUAL mode if acceptable
IF ctrl.eCtrlMode = E_METIS_CTRL_MODE.AUTO AND stat.bAcceptCtrlMode_Auto THEN
    stat.eCtrlMode := E_METIS_CTRL_MODE.AUTO;
ELSIF ctrl.eCtrlMode = E_METIS_CTRL_MODE.MANUAL AND stat.bAcceptCtrlMode_Manual THEN
    stat.eCtrlMode := E_METIS_CTRL_MODE.MANUAL;
END_IF

// switch to engineering ON / OFF mode if acceptable
stat.bEngMode := ctrl.bEngMode;

// switch to manual in any case if the input value is invalid
fbInputTimer(
    IN := (stat.eCtrlMode = E_METIS_CTRL_MODE.AUTO)
          AND (NOT pInputTemp^.stat.bValid),
    PT := DINT_TO_TIME(cfg.nInputTempTimeout));
fbSetpointTimer(
    IN := (stat.eCtrlMode = E_METIS_CTRL_MODE.AUTO)
           AND (NOT pSetpointTemp^.stat.bValid)
           AND cfg.eSetpointSwitch = E_METIS_CTRL_SETPOINT_SWITCH.VARIABLE,
    PT := DINT_TO_TIME(cfg.nSetpointTempTimeout)); 

IF fbInputTimer.Q OR fbSetpointTimer.Q THEN
    // calculate current time here, to avoid dependencies to MAIN.fbServices
    fbGetSystemTime(timeLoDW=>fileTime.dwLowDateTime, timeHiDW=>fileTime.dwHighDateTime );
    stat.sLastForcedManualTime := SYSTEMTIME_TO_STRING(FILETIME_TO_SYSTEMTIME(fileTime));
    IF fbInputTimer.Q THEN
        stat.sLastForcedManualCause := 'Invalid input temperature';
    ELSIF fbSetpointTimer.Q THEN
        stat.sLastForcedManualCause := 'Invalid setpoint temperature';
    ELSE
        stat.sLastForcedManualCause := 'UNKNOWN';
	END_IF
    
    stat.eCtrlMode := E_METIS_CTRL_MODE.MANUAL;
END_IF

// reset any request
ctrl.eCtrlMode := E_METIS_CTRL_MODE.NONE;
END_METHOD

METHOD M_GenerateRampedSetpoint : LREAL
VAR_INPUT
    in_bEnable                     : BOOL;
    in_bRestart                    : BOOL;

    in_lrTargetSetpoint            : LREAL;
    in_lrProcessValue              : LREAL;

    // Ramp rates in K/min
    in_lrRampUpRate                : LREAL;
    in_lrRampDownRate              : LREAL;

    // Maximum permitted difference between ramped SP and process value
    in_lrMaxTrackingDifference     : LREAL ;

    // A target step larger than this restarts the ramp from the process value
    in_lrTargetChangeThreshold     : LREAL;

    in_tCycleTime                  : TIME := T#10ms;
END_VAR

VAR_INST
    lrRampedSetpoint               : LREAL;
    lrPreviousTarget               : LREAL;

    bInitialized                   : BOOL;
    bWasEnabled                    : BOOL;
END_VAR

VAR
    lrCandidate                    : LREAL;
    lrRampUpStep                   : LREAL;
    lrRampDownStep                 : LREAL;
    lrTrackingLimit                : LREAL;
    lrTargetChangeThreshold        : LREAL;

    bTargetChanged                 : BOOL;
END_VAR
// Sanitize configuration values
lrTrackingLimit := ABS(in_lrMaxTrackingDifference);
lrTargetChangeThreshold := ABS(in_lrTargetChangeThreshold);


// Convert K/min into the increment for this PLC cycle.
// TIME_TO_LREAL returns the TIME value in milliseconds.
lrRampUpStep :=
    MAX(0.0, in_lrRampUpRate)
    * TIME_TO_LREAL(in_tCycleTime)
    / 60000.0;

lrRampDownStep :=
    MAX(0.0, in_lrRampDownRate)
    * TIME_TO_LREAL(in_tCycleTime)
    / 60000.0;


// Detect a meaningful target step.
// Small continuously moving targets do not repeatedly reset the ramp.
bTargetChanged :=
    bInitialized
    AND (
        ABS(in_lrTargetSetpoint - lrPreviousTarget)
        > lrTargetChangeThreshold
    );


// When disabled, synchronize with the process value.
// The next enable starts cleanly from the current temperature.
IF NOT in_bEnable THEN
    lrRampedSetpoint := in_lrProcessValue;
    lrPreviousTarget := in_lrTargetSetpoint;

    bInitialized := FALSE;
    bWasEnabled := FALSE;

    M_GenerateRampedSetpoint := lrRampedSetpoint;
    RETURN;
END_IF;


// Initialize or restart from the current process temperature.
IF NOT bInitialized
    OR NOT bWasEnabled
    OR in_bRestart
    OR bTargetChanged
THEN
    lrRampedSetpoint := in_lrProcessValue;
    bInitialized := TRUE;
END_IF;


// Remember the current command for the next cycle.
lrPreviousTarget := in_lrTargetSetpoint;
bWasEnabled := TRUE;


// Generate the normal time-based ramp candidate.
IF in_lrTargetSetpoint > lrRampedSetpoint THEN

    // Ramping upward
    lrCandidate :=
        MIN(
            in_lrTargetSetpoint,
            lrRampedSetpoint + lrRampUpStep
        );

ELSIF in_lrTargetSetpoint < lrRampedSetpoint THEN

    // Ramping downward
    lrCandidate :=
        MAX(
            in_lrTargetSetpoint,
            lrRampedSetpoint - lrRampDownStep
        );

ELSE
    lrCandidate := in_lrTargetSetpoint;
END_IF;


// Apply process-following constraint while heating.
//
// Only constrain when the target is above the actual process value.
// This avoids interfering with correction after an overshoot.
IF (in_lrTargetSetpoint > in_lrProcessValue)
    AND (
        lrCandidate
        > in_lrProcessValue + lrTrackingLimit
    )
THEN
    lrCandidate :=
        in_lrProcessValue + lrTrackingLimit;
END_IF;


// Apply process-following constraint while cooling.
//
// Only constrain when the target is below the actual process value.
IF (in_lrTargetSetpoint < in_lrProcessValue)
    AND (
        lrCandidate
        < in_lrProcessValue - lrTrackingLimit
    )
THEN
    lrCandidate :=
        in_lrProcessValue - lrTrackingLimit;
END_IF;


// Ensure the tracking constraint has not moved the generated value
// beyond the final target.
IF in_lrTargetSetpoint >= in_lrProcessValue THEN
    lrRampedSetpoint :=
        MIN(lrCandidate, in_lrTargetSetpoint);
ELSE
    lrRampedSetpoint :=
        MAX(lrCandidate, in_lrTargetSetpoint);
END_IF;


M_GenerateRampedSetpoint := lrRampedSetpoint;
END_METHOD

METHOD M_Read_Write_Config
VAR_IN_OUT
    temperatures : FB_NOTT_TEMPERATURES;
END_VAR
IF stat.bEngMode THEN
    IF ctrl.bWriteConfig THEN
        
        // update the cfg object
        cfg.sInputTempName      := pInputTemp^.in_sName;
        cfg.sSetpointTempName   := pSetpointTemp^.in_sName;
        cfg.lrFixedSetpoint     := ctrl.lrFixedSetpoint;
        cfg.lrSetpointOffset    := ctrl.lrSetpointOffset; 
        cfg.lrManualOut         := ctrl.lrManualOut;
        
        // write the cfg object
        fbTcConfig.M_WriteConfiguration();
        ctrl.bWriteConfig := FALSE;
                
    ELSIF ctrl.bReadConfig THEN
	
        fbTcConfig.M_ReadConfiguration();
        ctrl.bReadConfig := FALSE;
        
    END_IF
		
END_IF

IF fbTcConfig.bReadingDoneFlag THEN
	M_ConfigReadingFinished(
        bError := fbTcConfig.bReadError,
        temperatures := temperatures);
END_IF
END_METHOD

METHOD M_Set_SetPoint
VAR_INPUT
	m_eSetpointType:		E_METIS_CTRL_SETPOINT_SWITCH:=E_METIS_CTRL_SETPOINT_SWITCH.FIXED;
	m_pSetpointTemp: 		POINTER TO FB_METIS_TEMPERATURE;
	m_lrSetpointOffset: 	LREAL := 0.0;
	m_lrFixedSetpoint:	LREAL;
END_VAR

// Set point type 
cfg.eSetpointSwitch := m_eSetpointType;
// Variable setpoint
stat.lrActVariableSetpoint := m_pSetpointTemp^.stat.lrTempK;
ctrl.lrSetpointOffset:= m_lrSetpointOffset;
// Fixed setpoint
ctrl.lrFixedSetpoint := m_lrFixedSetpoint;
END_METHOD

METHOD M_SetDisable
VAR_INPUT
END_VAR

cfg.bEnabled := FALSE;
ctrl.eCtrlMode := E_METIS_CTRL_MODE.MANUAL;
END_METHOD

METHOD M_SetEnable
VAR_INPUT
END_VAR


cfg.bEnabled := TRUE;
ctrl.eCtrlMode := E_METIS_CTRL_MODE.AUTO;
END_METHOD

METHOD M_Startup : BOOL
VAR_INPUT
END_VAR
VAR_INST
	{attribute 'OPC.UA.DA' := '0'}
    startupTimer : TON;
END_VAR
startupTimer(IN := TRUE, PT := DINT_TO_TIME(cfg.nStartupTimeout));

IF NOT stat.bStarted THEN
    
    IF startupTimer.Q 
       OR (pInputTemp^.stat.bValid
           AND (pSetpointTemp^.stat.bValid 
                OR cfg.eSetpointSwitch = E_METIS_CTRL_SETPOINT_SWITCH.FIXED)) THEN
        stat.bStarted := TRUE; 
    END_IF
END_IF
END_METHOD

METHOD M_UpdateAlarms
VAR_INPUT
END_VAR
VAR
	stEventEntry : TcEventEntry;
	sText : STRING;
END_VAR
//
// Set / clear alarms
//

// Input temperature / process variable is invalid.
fbAlarmHandler.M_UpdateAlarm(
    in_bCondition    := cfg.bEnabled
                        AND stat.bStarted
                        AND (ctrl.nInputTempIndex <> 0)
                        AND (NOT stat.bActInputValid),
    in_nIndex        := 0,
    in_strEventEntry := Tc_Events.METISCryoPIDCtrlEventClass.InputTemperatureInvalid
);


// Variable setpoint temperature is invalid.
fbAlarmHandler.M_UpdateAlarm(
    in_bCondition    := cfg.bEnabled
                        AND stat.bStarted
                        AND (cfg.eSetpointSwitch = E_METIS_CTRL_SETPOINT_SWITCH.VARIABLE)
                        AND (ctrl.nSetpointTempIndex <> 0)
                        AND (NOT stat.bActVariableSetpointValid),
    in_nIndex        := 1,
    in_strEventEntry := Tc_Events.METISCryoPIDCtrlEventClass.VariableSetpointInvalid
);


// Controller was forced to manual mode.
fbAlarmHandler.M_UpdateAlarm(
    in_bCondition    := cfg.bEnabled
                        AND stat.bStarted
                        AND stat.bCtrlModeIsManual
                        AND (stat.sLastForcedManualCause <> ''),
    in_nIndex        := 2,
    in_strEventEntry := Tc_Events.METISCryoPIDCtrlEventClass.ControllerForcedManual
);


// PID function block error.
fbAlarmHandler.M_UpdateAlarm(
    in_bCondition    := cfg.bEnabled
                        AND stat.bStarted
                        AND fbCtrlPid.bError,
    in_nIndex        := 3,
    in_strEventEntry := Tc_Events.METISCryoPIDCtrlEventClass.PidBlockError
);


// Ramp function block error.
fbAlarmHandler.M_UpdateAlarm(
    in_bCondition    := cfg.bEnabled
                        AND stat.bStarted
                        AND ramp.stat.bError,
    in_nIndex        := 4,
    in_strEventEntry := Tc_Events.METISCryoPIDCtrlEventClass.RampBlockError
);


//
// Handle alarms
//
fbAlarmHandler(stAlarms := stat.stAlarms);

fbAlarmHandler.M_ProcessAlarms(
    arrEventEntry := arrEventEntry,
    sEventString  := in_sName
);
END_METHOD

METHOD M_UpdateStatus
VAR_INPUT
END_VAR
ctrl.nInputTempIndex := TO_INT(ctrl.eInputTempIndex);
ctrl.nSetpointTempIndex := TO_INT(ctrl.eVariableSetpointIndex);

// Alarm Handeling
sInstanceName := fbAlarmHandler.sInstanceName;
sEventClassName := fbAlarmHandler.sEventClassName;
IF bConfirmAllAlarms THEN
	bConfirmAllAlarms := FALSE;
	fbAlarmHandler.M_ConfirmAllAlarms();
END_IF

// update some more stat variables
stat.bSetpointSwitchIsFixed := cfg.eSetpointSwitch = E_METIS_CTRL_SETPOINT_SWITCH.FIXED;
stat.bSetpointSwitchIsVariable := cfg.eSetpointSwitch = E_METIS_CTRL_SETPOINT_SWITCH.VARIABLE;
stat.bCtrlModeIsAuto := stat.eCtrlMode = E_METIS_CTRL_MODE.AUTO;
stat.bCtrlModeIsManual := stat.eCtrlMode = E_METIS_CTRL_MODE.MANUAL;
stat.bActInputValid := (ctrl.nInputTempIndex <> 0) AND pInputTemp^.stat.bValid;
stat.bActVariableSetpointValid := (ctrl.nSetpointTempIndex <> 0) AND pSetpointTemp^.stat.bValid;

// update the textual status, and the bError and bWarning flags
IF NOT cfg.bEnabled THEN
    stat.sStatus := 'Disabled';
    stat.bError := FALSE;
ELSIF NOT stat.bStarted THEN
    stat.sStatus := 'Initializing';
ELSIF ctrl.nInputTempIndex = 0 THEN
    stat.sStatus := 'No input temperature configured';
    stat.bError := TRUE;
ELSIF NOT pInputTemp^.stat.bValid THEN
    stat.sStatus := 'Invalid input temperature';
    stat.bError := TRUE;
ELSIF      cfg.eSetpointSwitch = E_METIS_CTRL_SETPOINT_SWITCH.VARIABLE 
       AND ctrl.nSetpointTempIndex = 0 THEN
    stat.sStatus := 'No variable setpoint configured';
    stat.bError := TRUE;
ELSIF      cfg.eSetpointSwitch = E_METIS_CTRL_SETPOINT_SWITCH.VARIABLE 
       AND NOT pSetpointTemp^.stat.bValid THEN
    stat.sStatus := 'Invalid variable setpoint';
    stat.bError := TRUE;
ELSIF fbCtrlPid.bError THEN
    stat.sStatus := CONCAT('PID block error ', INT_TO_STRING(TO_INT(fbCtrlPid.eErrorId)));
    stat.bError := TRUE;
ELSIF ramp.stat.bError THEN
    stat.sStatus := CONCAT('Ramp block error ', INT_TO_STRING(TO_INT(ramp.stat.eErrorId)));
    stat.bError := TRUE;
ELSIF stat.eCtrlMode = E_METIS_CTRL_MODE.MANUAL THEN
    stat.bError := FALSE;
    stat.bWarning := FALSE;
    IF stat.bEngMode THEN
        stat.sStatus := 'MANUAL (ENG MODE)';
    ELSE
        stat.sStatus := 'MANUAL';
	END_IF
ELSIF stat.eCtrlMode = E_METIS_CTRL_MODE.AUTO THEN
    stat.bError := FALSE;
    stat.bWarning := FALSE;
    IF stat.bEngMode THEN
        stat.sStatus := 'AUTO (ENG MODE)';
    ELSE
        stat.sStatus := 'AUTO';
	END_IF
ELSE
    stat.bError := FALSE;
    stat.bWarning := TRUE;
    stat.sStatus := 'UNKNOWN STATUS';
END_IF

stat.bValid := NOT (stat.bError OR stat.bWarning);
END_METHOD

METHOD M_UpdateTempPointers
VAR_INPUT
END_VAR
VAR_IN_OUT
    temperatures : FB_NOTT_TEMPERATURES;
END_VAR
VAR 
    i : INT;
END_VAR
pInputTemp    := temperatures.all_temperatures[ctrl.nInputTempIndex];
pSetpointTemp := temperatures.all_temperatures[ctrl.nSetpointTempIndex];
END_METHOD

END_FUNCTION_BLOCK

// ---- POUs/Devices/Temp_voters/FB_NOTT_VOTERS.TcPOU
FUNCTION_BLOCK FB_NOTT_VOTERS
VAR_INPUT
END_VAR
VAR_OUTPUT
END_VAR
VAR_IN_OUT
	{attribute 'OPC.UA.DA' := '0'}
    nott_temp : FB_NOTT_TEMPERATURES;
END_VAR
VAR
	ctrl		: T_METIS_TEMP_VOTERS_CTRL;
	
	// SideCar  
	{attribute 'TcHmiSymbol.Show'}
    vote_sidecar  : FB_NOTT_VOTER;

	// Photonic Chip 
	{attribute 'TcHmiSymbol.Show'}
    vote_photonic_chip  : FB_NOTT_VOTER;	
	
	// Base Plate
	{attribute 'TcHmiSymbol.Show'}
    vote_base_plate  : FB_NOTT_VOTER;	
	
	// Shield
	{attribute 'TcHmiSymbol.Show'}
    vote_shield  : FB_NOTT_VOTER;	
	
	// Detector 
	{attribute 'TcHmiSymbol.Show'}
    vote_detector  : FB_NOTT_VOTER;
		
	// System temperatures
		{attribute 'TcHmiSymbol.Show'}
	vote_master_temp	: FB_NOTT_VOTER;
		{attribute 'TcHmiSymbol.Show'}
	vote_master_1		: FB_NOTT_VOTER;
		{attribute 'TcHmiSymbol.Show'}
	vote_master_2		: FB_NOTT_VOTER;
	
// Flat Field
		{attribute 'TcHmiSymbol.Show'}
	vote_flat_field:				FB_NOTT_VOTER;
		
// Thermal Box
	{attribute 'TcHmiSymbol.Show'}
	vote_thermal_box:				FB_NOTT_VOTER;	

// Cabinet
	{attribute 'TcHmiSymbol.Show'}
	vote_cabinet:					FB_NOTT_VOTER;	

//////////////////////////////////////////////////////////
// temperature Overide

    tor_vote_sidecar  :				FB_CRYO_CMD_OVERRIDE;
	bSim_Temp_vote_sidecar  :		BOOL := FALSE;	

END_VAR

	// SideCar  
vote_sidecar		(in_sName  := 'vote_sidecar', 		nott_temp := nott_temp);
	// Photonic Chip
vote_photonic_chip	(in_sName  := 'vote_photonic_chip', nott_temp := nott_temp);
	// Base Plate
vote_base_plate		(in_sName  := 'vote_base_plate', 	nott_temp := nott_temp);
	// Shield
vote_shield			(in_sName  := 'vote_shield', 		nott_temp := nott_temp);
	// Detector 
vote_detector(		in_sName  := 'vote_detector', 		nott_temp := nott_temp);

	// System temperatures
vote_master_temp(in_sName := 'MASTER_TEMP',   nott_temp := nott_temp);
vote_master_1(in_sName    := 'VOTE_MASTER_1', nott_temp := nott_temp);
vote_master_2(in_sName    := 'VOTE_MASTER_2', nott_temp := nott_temp);//, aTempIndexes := aVoteCry1TempIndexes, nVoteMethod := eVoteCry1Method, bEnabled := bEnableVoteCry1);

// Flat Field

vote_flat_field(in_sName    := 'vote_flat_field', nott_temp := nott_temp);

// Thermal Box

vote_thermal_box(in_sName    := 'vote_thermal_box', nott_temp := nott_temp);

// Cabinet

vote_cabinet(in_sName    := 'vote_cabinet', nott_temp := nott_temp);


M_ReadSensors();

M_ProcessHmi();

METHOD M_ProcessHmi : BOOL
VAR_INPUT
END_VAR
// hmi_temp_vote_cry_1(
// 	inout_sTemperatureStatRef 	:= vote_cry_1.stat,
// 	inout_sCmdOver 				:= ctrl.tor_vote_cry_1,
// 	inout_fbAlarmHandlerRef 	:= vote_cry_1.fbAlarmHandler,
// //	TestIndexes := TestIndexes, TestMethod := TestMethod
// );
END_METHOD

METHOD M_ReadSensors : BOOL
VAR_INPUT
END_VAR
//
// Read temperature votes.
//
// Execute Temperature Override (tor) of simulation flags.
tor_vote_sidecar(in_bEnable:=bSim_Temp_vote_sidecar);
END_METHOD

END_FUNCTION_BLOCK

// ---- POUs/Devices/Temp_voters/FB_NOTT_VOTER.TcPOU
FUNCTION_BLOCK FB_NOTT_VOTER
VAR_INPUT
	{attribute 'OPC.UA.DA' := '0'}
	in_sName:	STRING;
// 	{attribute 'OPC.UA.DA' := '0'}
// 	in_bSimulation	: BOOL;
	{attribute 'OPC.UA.DA' := '0'}
	in_nRampPeriodSec:		UDINT := 60;	// Ramp measurement period [sec]. Default 60 sec.
END_VAR
VAR_IN_OUT
	{attribute 'OPC.UA.DA' := '0'}
	nott_temp: FB_nott_TEMPERATURES;
END_VAR
VAR
	cfg:				T_NOTT_TEMP_VOTE_CFG;
// 	{attribute 'OPC.UA.DA' := '0'}
// 	bSimulation	: BOOL := FALSE;	// Simulated temp value

	{attribute 'OPC.UA.DA' := '0'}
	aTempPointers:	    ARRAY[0..4] OF POINTER TO FB_METIS_TEMPERATURE;
	{attribute 'OPC.UA.DA' := '0'}
	aTempIndexes:		ARRAY[0..4] OF INT := [0, 0, 0, 0, 0];
	
	(*Voting Method*)
	nVoteMethod:	E_METIS_TEMP_VOTE_METHOD := E_METIS_TEMP_VOTE_METHOD.AVERAGE;

	{attribute 'TcHmiSymbol.Show'}
	{attribute 'OPC.UA.DA' := '1'}
	stat	: T_NOTT_CRYO_TEMP_VOTE_STATUS;
    
    (* OLD PLC_HMI  *)
	{attribute 'TcHmiSymbol.Show'}
    bPLC_HMI:       BOOL := FALSE;
    
    (* User description *)
    //sDescription:   STRING;
    
	(*Engineering MODE*)
	{attribute 'TcHmiSymbol.Show'}
	bEngMode:		BOOL := FALSE;
	{attribute 'TcHmiSymbol.Show'}
	bAutoMode:		BOOL := TRUE;
	{attribute 'TcHmiSymbol.Show'}
	bManualMode:	BOOL := FALSE;	

	(*Configuration*)
	bConfigured:	BOOL := FALSE;
	
	(*Read/Write configuration*)
	{attribute 'OPC.UA.DA' := '0'}
	{attribute 'TcHmiSymbol.Show'}
	fbTempVoteConfig:		FB_NOTT_READ_WRITE_TEMP_VOTE_CONFIG;
	{attribute 'TcHmiSymbol.Show'}
	bReadConfig:			BOOL;
	{attribute 'TcHmiSymbol.Show'}	
	bWriteConfig:			BOOL;
	(*Ramp *)
	{attribute 'OPC.UA.DA' := '0'}
	bRampTimerStarted:	BOOL := FALSE;
	{attribute 'OPC.UA.DA' := '0'}
	rampTimer:	TON;		// Timer for calculating ramp
	
    // outputs that can be used for linking
	{attribute 'OPC.UA.DA' := '0'}
    q_lrTemp    AT %Q*: LREAL;
	{attribute 'OPC.UA.DA' := '0'}
	q_bToggle   AT %Q*: BOOL;
	{attribute 'OPC.UA.DA' := '0'}
	q_bValid   AT %Q*: BOOL := FALSE;
	
	{attribute 'TcHmiSymbol.Show'}
	{attribute 'TcHmiSymbol.ReadOnly'}
	sEventClassName : T_MaxString;


	{attribute 'TcHmiSymbol.Show'}
	bConfirmAllAlarms : BOOL;
	
		// Alarm handling
	// List of alarms to be handled by Temperature
	arrEventEntry : ARRAY [0..5] OF TcEventEntry;
	// Alarm handler FB

	fbAlarmHandler : FB_AlarmHandler;
	{attribute 'TcHmiSymbol.Show'}
	{attribute 'TcHmiSymbol.ReadOnly'}
	sInstanceName : T_MaxString := fbAlarmHandler.sInstanceName;
	// Logs logs
	logs:	FB_CRYO_FUNCTION_LOG;
END_VAR

// to avoid any problem of invalid pointers, set them right away
M_UpdateTempPointers(nott_temp := nott_temp);

(*Read/Write configuration*)
fbTempVoteConfig(in_sTVoteName:= in_sName, Temp_Vote_Config:= cfg);

IF NOT bConfigured THEN
    M_Configure(nott_temp := nott_temp);
    RETURN;
END_IF

// set AUTO / MAN / ENG
M_SetPermissionMode();

// read/write the config (if needed)
M_Read_Write_Config(nott_temp := nott_temp);

M_GetRamp();

M_SetStatus();


// Handle alarms
M_UpdateAlarms();

PROPERTY bTempNotValid : BOOL
GET
bTempNotValid := NOT stat.bValid;
END_GET
END_PROPERTY

PROPERTY bTempValid : BOOL
GET
bTempValid := stat.bValid;
END_GET
END_PROPERTY

PROPERTY lrRamp : LREAL
GET
lrRamp := stat.lrRamp;
END_GET
END_PROPERTY

PROPERTY lrTempK : LREAL
GET
lrTempK := stat.lrTempK;
END_GET
END_PROPERTY

METHOD M_ConfigReadingFinished
VAR_INPUT
    bError : BOOL;
END_VAR
VAR_IN_OUT
    nott_temp : FB_NOTT_TEMPERATURES;
END_VAR
VAR
    i : INT;
END_VAR
IF bError THEN
   // ERROR! Just put the indexes to 0
   FOR i := 0 TO 4 DO
       aTempIndexes[i] := 0;
   END_FOR
   stat.bEnabled := FALSE;
   stat.sDescription := in_sName;
ELSE
    // success!
//     aTempIndexes[0] := met_temp.M_GetTempSensorIndex(cfg.sTemp1_Name);
//     aTempIndexes[1] := met_temp.M_GetTempSensorIndex(cfg.sTemp2_Name);
//     aTempIndexes[2] := met_temp.M_GetTempSensorIndex(cfg.sTemp3_Name);
//     aTempIndexes[3] := met_temp.M_GetTempSensorIndex(cfg.sTemp4_Name);
//     aTempIndexes[4] := met_temp.M_GetTempSensorIndex(cfg.sTemp5_Name);
// 	aTempIndexes[0] 	:= TO_INT(cfg.eTemperature1);
// 	aTempIndexes[1] 	:= TO_INT(cfg.eTemperature2);
// 	aTempIndexes[2] 	:= TO_INT(cfg.eTemperature3);
// 	aTempIndexes[3] 	:= TO_INT(cfg.eTemperature4);
// 	aTempIndexes[4] 	:= TO_INT(cfg.eTemperature5);
    stat.nVoteMethod     := cfg.nVote_Method;
    stat.bEnabled        := cfg.bEnabled;
    stat.sDescription    := cfg.sDescription;
	stat.aTempIndexes[0] := cfg.eTemperature1;
	stat.aTempIndexes[1] := cfg.eTemperature2;
    stat.aTempIndexes[2] := cfg.eTemperature3;
	stat.aTempIndexes[3] := cfg.eTemperature4;
    stat.aTempIndexes[4] := cfg.eTemperature5; 
END_IF

M_UpdateTempPointers(nott_temp := nott_temp);

// clear the flag
fbTempVoteConfig.M_ClearReadingDoneFlag();
END_METHOD

METHOD M_Configure : BOOL
VAR_INPUT
END_VAR
VAR_INST
	{attribute 'OPC.UA.DA' := '0'}
    nConfigureState : INT;
END_VAR
VAR_IN_OUT
	{attribute 'OPC.UA.DA' := '0'}
    nott_temp : FB_NOTT_TEMPERATURES;
END_VAR
VAR
    i : INT;
END_VAR











CASE nConfigureState OF
    0:  
        // use the name of the voter as the default description
        stat.sDescription := in_sName;
        // start reading the config
        fbTempVoteConfig.M_ReadConfiguration();
        nConfigureState := 1;
    1:
        IF fbTempVoteConfig.bReadingDoneFlag THEN
            M_ConfigReadingFinished(
                bError   := fbTempVoteConfig.bReadError,
                nott_temp := nott_temp);
		
			//
	// Populate array of Alarms.
	//
	// See the definition of CryoPressVoteEventClass under Type System.
	//
	arrEventEntry[0] := Tc_Events.METISCryoTempEventClass.ReadingNotValid;
	arrEventEntry[1] := Tc_Events.METISCryoTempEventClass.Sensor1Error;
	arrEventEntry[2] := Tc_Events.METISCryoTempEventClass.Sensor2Error;
	arrEventEntry[3] := Tc_Events.METISCryoTempEventClass.Sensor3Error;
	arrEventEntry[4] := Tc_Events.METISCryoTempEventClass.Sensor4Error;
	arrEventEntry[5] := Tc_Events.METISCryoTempEventClass.Sensor5Error;
            
            bConfigured := TRUE;
        END_IF
END_CASE
END_METHOD

METHOD M_GetRamp
VAR_INPUT
END_VAR
VAR_INST
	{attribute 'OPC.UA.DA' := '0'}
	lrRampStartTempK:	LREAL;	// Temperature at start of ramp timer [K]
END_VAR
VAR
	nRampPeriodSec:		UDINT;	// Ramp measurement period [sec].
END_VAR

IF NOT (stat.bEnabled AND stat.bValid) THEN
    bRampTimerStarted := FALSE;
    stat.lrRamp := 0.0;
    RETURN;
END_IF

IF NOT bRampTimerStarted THEN
	bRampTimerStarted	:= TRUE;
	lrRampStartTempK	:= stat.lrTempK;
	rampTimer(IN:=FALSE);
END_IF

// Execute timer.
// Ramp measurement period should be > 0
nRampPeriodSec	:= in_nRampPeriodSec;
IF nRampPeriodSec = 0 THEN
	nRampPeriodSec	:= 60;
END_IF
rampTimer(IN:=TRUE,PT:=UDINT_TO_TIME(nRampPeriodSec)*1000);

// Calculate ramp at time expiry
IF rampTimer.Q THEN
	// Calculate the temperature ramp per minute
//	IF stat.bValid THEN
		stat.lrRamp	:= (stat.lrTempK - lrRampStartTempK) * 60.0 / nRampPeriodSec;
//	ELSE
//		stat.lrRamp	:= 0.0;
//	END_IF

	// Current temperature is the starting value of the ramp
	lrRampStartTempK	:= stat.lrTempK;

	// Restart the timer
	rampTimer(IN:=FALSE);
END_IF
END_METHOD

METHOD M_Read_Write_Config
VAR_INPUT
END_VAR
VAR_IN_OUT
    nott_temp : FB_NOTT_TEMPERATURES;
END_VAR
IF bEngMode THEN
    IF bWriteConfig THEN
        
        // update the cfg object
        cfg.bEnabled     := stat.bEnabled;
        cfg.sDescription := stat.sDescription;
        cfg.sTemp1_Name  := aTempPointers[0]^.in_sName;
        cfg.sTemp2_Name  := aTempPointers[1]^.in_sName; 
        cfg.sTemp3_Name  := aTempPointers[2]^.in_sName; 
        cfg.sTemp4_Name  := aTempPointers[3]^.in_sName; 
        cfg.sTemp5_Name  := aTempPointers[4]^.in_sName;
        cfg.nVote_Method := stat.nVoteMethod;
		cfg.eTemperature1:= stat.aTempIndexes[0];
		cfg.eTemperature2:= stat.aTempIndexes[1];
		cfg.eTemperature3:= stat.aTempIndexes[2];
		cfg.eTemperature4:= stat.aTempIndexes[3];
		cfg.eTemperature5:= stat.aTempIndexes[4];
        
        // write the cfg object
        fbTempVoteConfig.M_WriteConfiguration();
        bWriteConfig := FALSE;
                
    ELSIF bReadConfig THEN
	
        fbTempVoteConfig.M_ReadConfiguration();
        bReadConfig := FALSE;
        
    END_IF
		
END_IF

IF fbTempVoteConfig.bReadingDoneFlag THEN
	M_ConfigReadingFinished(
        bError := fbTempVoteConfig.bReadError,
        nott_temp := nott_temp);
END_IF
END_METHOD

METHOD M_SetPermissionMode : BOOL
VAR_INPUT
END_VAR
IF bAutoMode THEN
    stat.sStatus    := 'AUTO';
    bManualMode     := FALSE;
    bEngMode        := FALSE;
ELSIF bEngMode	THEN
    stat.sStatus    := 'ENG';
    bManualMode     := FALSE;
    bAutoMode       := FALSE;
ELSIF bManualMode THEN
    stat.sStatus    := 'MANUAL';
    bAutoMode       := FALSE;
    bEngMode        := FALSE;
END_IF
END_METHOD

// Calculate pressure based on the status of the two sensors
METHOD M_SetStatus
VAR_INPUT
END_VAR
VAR
	lrTmp:		LREAL;	// Temporary var
	nSample:	INT;
	i:			INT;
END_VAR
VAR_INST
	{attribute 'OPC.UA.DA' := '0'}
    toggleTimer : TON;
END_VAR
aTempIndexes[0] 	:= TO_INT(stat.aTempIndexes[0]);
aTempIndexes[1] 	:= TO_INT(stat.aTempIndexes[1]);
aTempIndexes[2] 	:= TO_INT(stat.aTempIndexes[2]);
aTempIndexes[3] 	:= TO_INT(stat.aTempIndexes[3]);
aTempIndexes[4] 	:= TO_INT(stat.aTempIndexes[4]);


stat.lrSens1TempK := aTempPointers[0]^.stat.lrTempK;
stat.lrSens2TempK := aTempPointers[1]^.stat.lrTempK;
stat.lrSens3TempK := aTempPointers[2]^.stat.lrTempK;
stat.lrSens4TempK := aTempPointers[3]^.stat.lrTempK;
stat.lrSens5TempK := aTempPointers[4]^.stat.lrTempK;

stat.bValidSensor1  := aTempPointers[0]^.stat.bValid;
stat.bValidSensor2  := aTempPointers[1]^.stat.bValid;
stat.bValidSensor3  := aTempPointers[2]^.stat.bValid;
stat.bValidSensor4  := aTempPointers[3]^.stat.bValid;
stat.bValidSensor5  := aTempPointers[4]^.stat.bValid;

// copy some writeable values to the read-only stat struct
//stat.bEnabled := bEnabled;
//stat.sDescription := sDescription;

sInstanceName := fbAlarmHandler.sInstanceName;
sEventClassName := fbAlarmHandler.sEventClassName;
IF bConfirmAllAlarms THEN
	bConfirmAllAlarms := FALSE;
	fbAlarmHandler.M_ConfirmAllAlarms();
END_IF


// If disabled, don't do anything
IF NOT stat.bEnabled THEN
    stat.bValid := FALSE;
    RETURN;
END_IF

//
// If simulated, set the simulated value and return.
//
IF stat.bSimulated THEN
// 	stat.bSimulated	:= TRUE;
	stat.bValid		:= TRUE;
	stat.lrTempK	:= stat.lrSimTempK;
	RETURN;
ELSE
	stat.bSimulated	:= FALSE;
END_IF


//
// Get the pressure depending on the voting method.
//
CASE nVoteMethod OF
	E_METIS_TEMP_VOTE_METHOD.AVERAGE:
		M_SetStatus_Average();
	E_METIS_TEMP_VOTE_METHOD.LOWEST_TEMPERATURE:
		M_SetStatus_Lowest_Temperature();
	E_METIS_TEMP_VOTE_METHOD.HIGHEST_TEMPERATURE:
		M_SetStatus_Highest_Temperature();
	E_METIS_TEMP_VOTE_METHOD.FIRST_VALID_TEMPERATURE:
		M_SetStatus_FirstValid();
	E_METIS_TEMP_VOTE_METHOD.MEDIAN:
		M_SetStatus_Median();
//	E_METIS_TEMP_VOTE_METHOD.TEMPERATURE_3oo5:
//		M_SetStatus_XooY();
ELSE
	;
END_CASE


//
// If the reading is valid, set the simulated value to it.
// This way, switching from normal to simulation will result in
// no jump in the value.
//
IF stat.bValid  THEN
	stat.lrSimTempK	:= stat.lrTempK;
END_IF

// update also the output data
q_lrTemp := stat.lrTempK;
q_bValid := stat.bValid;
toggleTimer(IN := NOT toggleTimer.Q, PT := T#500ms);
IF toggleTimer.Q AND stat.bValid THEN
    q_bToggle := NOT q_bToggle;
END_IF
END_METHOD

METHOD M_SetStatus_Average
VAR_INPUT
END_VAR
VAR
	lrTmp:		LREAL;	// Temporary var for sum of Temperatures
	nSample:	INT;	// Number of valid sensor readings
	i:			INT;
END_VAR
lrTmp	:= 0.0;
nSample	:= 0;

FOR i:=0 TO 4 DO
	IF aTempIndexes[i] > 0  THEN
		IF aTempPointers[i]^.stat.bValid	THEN
			lrTmp	:= lrTmp + aTempPointers[i]^.stat.lrTempK;
			nSample	:= nSample + 1;
		END_IF
	END_IF
END_FOR

IF nSample > 0	THEN
	stat.lrTempK	:= lrTmp / nSample;
	stat.bValid		:= TRUE;
ELSE
	stat.lrTempK	:= 9999;
	stat.bValid		:= FALSE;
END_IF
END_METHOD

METHOD M_SetStatus_FirstValid
VAR_INPUT
END_VAR
VAR
	lrTmp:		LREAL;	// Temporary var for sum of Temperatures
	nSample:	INT;	// Number of valid sensor readings
	i:			INT;
END_VAR
(*First Valid Temperature*)

nSample	:= 0;

FOR i:=0 TO 4 DO
	IF aTempIndexes[i] > 0  THEN
		IF  aTempPointers[i]^.stat.bValid	THEN
			lrTmp	:= aTempPointers[i]^.stat.lrTempK;
			nSample	:= nSample + 1;
			EXIT;
		END_IF
	END_IF
END_FOR

IF nSample > 0	THEN
	stat.lrTempK	:= lrTmp;
	stat.bValid		:= TRUE;
ELSE
	stat.lrTempK	:= 9999;
	stat.bValid		:= FALSE;
END_IF
END_METHOD

METHOD M_SetStatus_Highest_Temperature
VAR_INPUT
END_VAR
VAR
	lrTmp:		LREAL;	// Temporary var for sum of Temperatures
	nSample:	INT;	// Number of valid sensor readings
	i:			INT;
END_VAR
(*Highest Temperature*)

lrTmp	:= -10000.0; // setting initial temperature for comparision
nSample	:= 0;

FOR i:=0 TO 4 DO
	IF aTempIndexes[i] > 0  THEN
		IF  aTempPointers[i]^.stat.bValid	THEN
				IF  aTempPointers[i]^.stat.lrTempK > lrTmp THEN
					lrTmp	:= aTempPointers[i]^.stat.lrTempK;
				END_IF
			nSample	:= nSample + 1;
		END_IF
	END_IF
END_FOR

IF nSample > 0	THEN
	stat.lrTempK	:= lrTmp;
	stat.bValid		:= TRUE;
ELSE
	stat.lrTempK	:= 9999;
	stat.bValid		:= FALSE;
END_IF
END_METHOD

METHOD M_SetStatus_Lowest_Temperature
VAR_INPUT
END_VAR
VAR
	lrTmp:		LREAL;	// Temporary var for sum of Temperatures
	nSample:	INT;	// Number of valid sensor readings
	i:			INT;
END_VAR
(*Lowest Temperature*)

lrTmp	:= 10000.0; // setting initial temperature for comparision
nSample	:= 0;

FOR i:=0 TO 4 DO
	IF aTempIndexes[i] > 0  THEN
		IF  aTempPointers[i]^.stat.bValid	THEN
				IF  aTempPointers[i]^.stat.lrTempK < lrTmp THEN
					lrTmp	:= aTempPointers[i]^.stat.lrTempK;
				END_IF
			nSample	:= nSample + 1;
		END_IF
	END_IF
END_FOR

IF nSample > 0	THEN
	stat.lrTempK	:= lrTmp;
	stat.bValid		:= TRUE;
ELSE
	stat.lrTempK	:= 9999;
	stat.bValid		:= FALSE;
END_IF
END_METHOD

METHOD M_SetStatus_Median
VAR_INPUT
END_VAR
VAR
    lrTmpArray: ARRAY[0..4] OF LREAL; // Array to store valid temperatures
    nSample:    INT;                // Number of valid sensor readings
    i:          INT;
    j:          INT;
    lrTemp:     LREAL;             // Temporary variable for swapping
END_VAR
nSample := 0;

// Store valid temperatures in the array
FOR i := 0 TO 4 DO
    IF aTempIndexes[i] > 0 THEN
        IF aTempPointers[i]^.stat.bValid THEN
            lrTmpArray[nSample] := aTempPointers[i]^.stat.lrTempK;
            nSample := nSample + 1;
        END_IF
    END_IF
END_FOR

// Sort the array in ascending order (using Bubble Sort for simplicity)
IF nSample > 1 THEN
    FOR i := 0 TO nSample - 2 DO
        FOR j := i + 1 TO nSample - 1 DO
            IF lrTmpArray[i] > lrTmpArray[j] THEN
                lrTemp := lrTmpArray[i];
                lrTmpArray[i] := lrTmpArray[j];
                lrTmpArray[j] := lrTemp;
            END_IF
        END_FOR
    END_FOR
END_IF

// Calculate the median
IF nSample > 0 THEN
    IF nSample MOD 2 = 1 THEN // Odd number of elements
        stat.lrTempK := lrTmpArray[nSample / 2];
    ELSE // Even number of elements
        stat.lrTempK := (lrTmpArray[nSample / 2 - 1] + lrTmpArray[nSample / 2]) / 2.0;
    END_IF
    stat.bValid := TRUE;
ELSE
    stat.lrTempK := 9999;
    stat.bValid := FALSE;
END_IF
END_METHOD

// Calculate pressure based on the status of the two sensors
METHOD M_SetStatus_XooY
//VAR_INPUT
//	in_nNum:	INT;	// Number of readings to select for voting (X)
//	in_nTotal:	INT;	// Total number of readings to check (Y)
//END_VAR
//VAR
//	idx_i, idx_j:	INT;
//	nTmp:		INT;			// Temporary INT var
//	lrTmp:		LREAL	:= 0.0;	// Temporary var for sum of pressures
//	nValid:		INT		:= 0;	// Total number of valid readings
//	nSample:	INT		:= 0;	// Number of valid sensor readings
	
//	aDiff:		ARRAY [1..5,1..5] OF LREAL;	// Table of absolute differences
//	aDiffSum:	ARRAY [1..5] OF LREAL;		// Array of sums of absolute differences
//	// Array of indexes of sums of absolute differences
//	aDiffSumIdx:ARRAY [1..5] OF INT := [1,2,3,4,5];		
//	lrAbsDiff:	LREAL;						// Absolute difference between two readings
	
//	i:			INT;
//	j:			INT;
//END_VAR
VAR
	lrTmp:		LREAL;	// Temporary var for sum of Temperatures
	nSample:	INT;	// Number of valid sensor readings
	i:			INT;
END_VAR
(*Average Temperature*)

lrTmp	:= 0.0;
nSample	:= 0;

FOR i:=0 TO 4 DO
	IF aTempIndexes[i] > 0  THEN
		IF  aTempPointers[i]^.stat.bValid	THEN
			lrTmp	:= lrTmp + aTempPointers[i]^.stat.lrTempK;
			nSample	:= nSample + 1;
		END_IF
	END_IF
END_FOR

IF nSample > 0	THEN
	stat.lrTempK	:= lrTmp / nSample;
	stat.bValid		:= TRUE;
ELSE
	stat.lrTempK	:= 9999;
	stat.bValid		:= FALSE;
END_IF








////
////	Get the number of valid readings and calculate the average
////
//FOR i:=1 TO in_nTotal DO
//	IF pSensor[i] <> 0  THEN
//		IF  pSensor[i]^.stat.bValid	THEN
//			lrTmp	:= lrTmp + pSensor[i]^.stat.lrPressure;
//			nValid	:= nValid + 1;
//		END_IF
//	END_IF
//END_FOR


////
//// Vote X out of Y
////
//IF nValid >= in_nNum	THEN
//	//
//	// Calculate relative differences between two readings, 
//	// relative to the bigger ABS value.
//	// Table is symetric. Calculate only the half (triangle) on the right. 
//	// Make a copy to the other half.
//	//
//	FOR i:=1 TO in_nTotal DO
//		FOR j:=i+1 TO in_nTotal DO
//			IF pSensor[i] <> 0  AND  pSensor[j] <> 0	THEN
//				IF pSensor[i]^.stat.bValid  AND  pSensor[j]^.stat.bValid	THEN
//					lrAbsDiff	:= ABS(pSensor[i]^.stat.lrPressure - pSensor[j]^.stat.lrPressure);
//					aDiff[i,j]	:= lrAbsDiff;
//					aDiff[j,i]	:= lrAbsDiff;
//				ELSE
//					aDiff[i,j]	:= 9999.0;
//					aDiff[j,i]	:= 9999.0;
//				END_IF
//			ELSE
//				aDiff[i,j]	:= 9999.0;
//				aDiff[j,i]	:= 9999.0;
//			END_IF
//		END_FOR
//	END_FOR

//	//
//	// Get the sum of all differences for each reading.
//	//
//	FOR i:=1 TO in_nTotal DO
//		aDiffSum[i]	:= 0.0;
//		FOR j:=1 TO in_nTotal DO
//			aDiffSum[i]	:= aDiffSum[i] + aDiff[i,j];
//		END_FOR
//	END_FOR

//	//
//	// Sort the indexes for differences in accending order (low sum first).
//	//
//	FOR i:=1 TO in_nTotal DO
//		FOR j:=i+1 TO in_nTotal DO
//			idx_i	:= aDiffSumIdx[i];
//			idx_j	:= aDiffSumIdx[j];
//			IF aDiffSum[idx_j] < aDiffSum[idx_i]	THEN
//				// Swap indexes
//				nTmp			:= aDiffSumIdx[j];
//				aDiffSumIdx[j]	:= aDiffSumIdx[i];
//				aDiffSumIdx[i]	:= nTmp;
//			END_IF
//		END_FOR
//	END_FOR

	
//	//					
//	// Get the average of selected in_nNum readings.
//	// Assign the result to the pressure.
//	//
//	lrTmp	:= 0.0;
//	FOR i:=1 TO in_nNum DO
//		idx_i	:= aDiffSumIdx[i];
//		lrTmp	:= lrTmp + pSensor[idx_i]^.stat.lrPressure;
//	END_FOR
	
//	stat.lrPressure	:= lrTmp / in_nNum;
//	stat.bValid		:= TRUE;
//ELSE
//	stat.lrPressure	:= 9999;
//	stat.bValid		:= FALSE;
//END_IF
END_METHOD

METHOD M_UpdateAlarms
VAR_INPUT
END_VAR
VAR
	stEventEntry : TcEventEntry;
	sText : STRING;
END_VAR
//
// Set / clear alarms
//

// Global alarm if the voted temperature reading is not valid.
fbAlarmHandler.M_UpdateAlarm(
    in_bCondition    := NOT stat.bValid,
    in_nIndex        := 0,
    in_strEventEntry := Tc_Events.METISCryoTempEventClass.ReadingNotValid
);


// Individual sensor alarms.
// Important:
// Even if aTempIndexes[x] = 0, M_UpdateAlarm is still called with FALSE.
// This ensures that any previously active alarm is cleared automatically.

fbAlarmHandler.M_UpdateAlarm(
    in_bCondition    := (aTempIndexes[0] > 0) AND (NOT aTempPointers[0]^.stat.bValid),
    in_nIndex        := 1,
    in_strEventEntry := Tc_Events.METISCryoTempEventClass.Sensor1Error
);

fbAlarmHandler.M_UpdateAlarm(
    in_bCondition    := (aTempIndexes[1] > 0) AND (NOT aTempPointers[1]^.stat.bValid),
    in_nIndex        := 2,
    in_strEventEntry := Tc_Events.METISCryoTempEventClass.Sensor2Error
);

fbAlarmHandler.M_UpdateAlarm(
    in_bCondition    := (aTempIndexes[2] > 0) AND (NOT aTempPointers[2]^.stat.bValid),
    in_nIndex        := 3,
    in_strEventEntry := Tc_Events.METISCryoTempEventClass.Sensor3Error
);

fbAlarmHandler.M_UpdateAlarm(
    in_bCondition    := (aTempIndexes[3] > 0) AND (NOT aTempPointers[3]^.stat.bValid),
    in_nIndex        := 4,
    in_strEventEntry := Tc_Events.METISCryoTempEventClass.Sensor4Error
);

fbAlarmHandler.M_UpdateAlarm(
    in_bCondition    := (aTempIndexes[4] > 0) AND (NOT aTempPointers[4]^.stat.bValid),
    in_nIndex        := 5,
    in_strEventEntry := Tc_Events.METISCryoTempEventClass.Sensor5Error
);


//
// Handle alarms
//
fbAlarmHandler(stAlarms := stat.stAlarms);

fbAlarmHandler.M_ProcessAlarms(
    arrEventEntry := arrEventEntry,
    sEventString  := in_sName
);
END_METHOD

METHOD M_UpdateTempPointers
VAR_INPUT
END_VAR
VAR_IN_OUT
    nott_temp : FB_NOTT_TEMPERATURES;
END_VAR
VAR 
    i : INT;
END_VAR
// FOR i := 0 TO 4 DO
//     aTempPointers[i] := met_temp.M_SetTemperatureSensor(aTempIndexes[i]);
// END_FOR

FOR i := 0 TO 4 DO
	IF bPLC_HMI THEN
	    aTempPointers[i] := nott_temp.M_SetTemperatureSensor(TO_INT(aTempIndexes[i]));
	ELSE	(*Temp selection from new HMI*)
    	aTempPointers[i] := nott_temp.M_SetTemperatureSensor(TO_INT(stat.aTempIndexes[i]));
	END_IF


END_FOR
END_METHOD

END_FUNCTION_BLOCK

// ---- POUs/Devices/Temp_voters/FB_NOTT_READ_WRITE_TEMP_VOTE_CONFIG.TcPOU
FUNCTION_BLOCK FB_NOTT_READ_WRITE_TEMP_VOTE_CONFIG EXTENDS FB_READ_WRITE_CONFIG_BASE
VAR_INPUT
	in_sTVoteName:      T_MaxString;
END_VAR
VAR_IN_OUT
	Temp_Vote_Config:   T_NOTT_TEMP_VOTE_CFG;
END_VAR

SUPER^(
    in_sEntryName  := in_sTVoteName,
    in_sSubFolder  := 'Temperature_Vote\',
    in_sXPath      := '/Temperature_Vote_Configuration/',
    in_pSymAddr    := ADR(Temp_Vote_Config),
    in_cbSymSize   := SIZEOF(Temp_Vote_Config));

END_FUNCTION_BLOCK

// ---- POUs/Routines/WarmUp/FB_NOTT_CRYO_WARMUP.TcPOU
FUNCTION_BLOCK FB_NOTT_CRYO_WARMUP
VAR_INPUT
	in_bEnable:	BOOL := FALSE;	// System active while in_bEnable is TRUE
	in_Cryo_Stat:	T_NOTT_CRYO_STAT;
END_VAR
VAR_OUTPUT
	out_bPermit_Evacuation_Stop:	BOOL := FALSE;
	out_bPermit_CoolDown:				BOOL := FALSE;
END_VAR
VAR_IN_OUT
	{attribute 'OPC.UA.DA' := '0'}
	nott_temps:						FB_NOTT_TEMPERATURES;
	{attribute 'OPC.UA.DA' := '0'}
	nott_heaters:					FB_NOTT_HEATERS;
	{attribute 'OPC.UA.DA' := '0'}
	nott_t_ctrls:      				FB_NOTT_TCTRLs;
	{attribute 'OPC.UA.DA' := '0'}
	nott_t_votes: 					FB_NOTT_VOTERS;
END_VAR
VAR
		
	{attribute 'TcHmiSymbol.Show'}	
	cfg:	T_NOTT_CRYO_WARMUP_CFG;
	{attribute 'TcHmiSymbol.Show'}
	ctrl:	T_NOTT_CRYO_WARMUP_CTRL;
	{attribute 'OPC.UA.DA' := '1'}
	{attribute 'TcHmiSymbol.Show'}
	stat:	T_NOTT_CRYO_WARMUP_STAT;
	
//
// Internals
//
	timer:	TON;
	trig:	R_TRIG;	// Start trigger
//

	{attribute 'TcHmiSymbol.Show'}
	bPermitStart:	BOOL := FALSE;
	{attribute 'TcHmiSymbol.Show'}
	bPermitStop:	BOOL := FALSE;
	
END_VAR

M_Configure();
M_ExecuteControllers();
M_SafetyCheck();
M_StateMachine( 
	nott_temps  := nott_temps,
	nott_heaters := nott_heaters,
	nott_t_ctrls := nott_t_ctrls,
	nott_t_votes := nott_t_votes
);
M_UpdateStatus();

METHOD M_Configure
VAR_INPUT
END_VAR
VAR
	refBOOL:	REFERENCE TO BOOL;
END_VAR
// IF stat.bConfigured THEN
// 
// ELSE
// 	RETURN;
// END_IF
END_METHOD

METHOD M_ExecuteControllers
VAR
	ptrSimTemp:	POINTER TO LREAL;
END_VAR
END_METHOD

METHOD M_PermitStart_WarmUp
VAR_INPUT
	in_bPermissionStart: BOOL;
END_VAR
bPermitStart := in_bPermissionStart;
END_METHOD

METHOD M_PermitStop_WarmUp
VAR_INPUT
	in_bPermissionStop: BOOL;
END_VAR
bPermitStop := in_bPermissionStop;
END_METHOD

METHOD M_SafetyCheck
VAR_INPUT
END_VAR
VAR CONSTANT
	lrPress_WarmAlarmTrip:	LREAL := 10.0E-1;	// [mbar]
	lrPress_WarmAlarmReset:	LREAL := 8.0E-1;	// [mbar], hysteresis reset
END_VAR
// Keep pressure and pump alarm causes separate so clearing one condition
// cannot hide the other.
IF NOT stat.bActive THEN
	stat.bPressureAlarm := FALSE;
ELSIF in_Cryo_Stat.bPressureValid THEN
	IF stat.bPressureAlarm THEN
		IF in_Cryo_Stat.lrPressure_mbar < lrPress_WarmAlarmReset THEN
			stat.bPressureAlarm := FALSE;
		END_IF
	ELSIF in_Cryo_Stat.lrPressure_mbar > lrPress_WarmAlarmTrip THEN
		stat.bPressureAlarm := TRUE;
	END_IF
END_IF

// A pump loss during active warmup disables every heat source and trips the
// routine. The alarm resets only after both pumps recover; restart is manual.
IF stat.bActive
	AND (NOT in_Cryo_Stat.bIsPVPRunning OR NOT in_Cryo_Stat.bIsTMPRunning) THEN
	stat.bPumpAlarm := TRUE;

	nott_heaters.h_detector.M_SetDisable();
	nott_heaters.h_detector_spare.M_SetDisable();
	nott_heaters.h_sidecar.M_SetDisable();
	nott_heaters.h_photonic_chip.M_SetDisable();
	nott_heaters.h_base_plate.M_SetDisable();
	nott_heaters.h_shield.M_SetDisable();

	nott_t_ctrls.tc_detector.M_SetDisable();
	nott_t_ctrls.tc_detector_spare.M_SetDisable();
	nott_t_ctrls.tc_sidecar.M_SetDisable();
	nott_t_ctrls.tc_photonic_chip.M_SetDisable();
	nott_t_ctrls.tc_base_plate.M_SetDisable();
	nott_t_ctrls.tc_shields.M_SetDisable();

	stat.nState := E_NOTT_CRYO_WARMUP_STATE.STOP_WARMUP;
	stat.sErrorText := 'Pump stopped during warmup.';
ELSIF in_Cryo_Stat.bIsPVPRunning AND in_Cryo_Stat.bIsTMPRunning THEN
	stat.bPumpAlarm := FALSE;
END_IF

stat.bAlarm := stat.bPressureAlarm OR stat.bPumpAlarm;
stat.bWarning := stat.bAlarm;
END_METHOD

METHOD M_StateMachine : BOOL
VAR_INPUT
END_VAR
VAR_IN_OUT
    {attribute 'OPC.UA.DA' := '0'}
    nott_temps   : FB_NOTT_TEMPERATURES;
    {attribute 'OPC.UA.DA' := '0'}
    nott_heaters : FB_NOTT_HEATERS;
    {attribute 'OPC.UA.DA' := '0'}
    nott_t_ctrls : FB_NOTT_TCTRLs;
    {attribute 'OPC.UA.DA' := '0'}
    nott_t_votes : FB_NOTT_VOTERS;
END_VAR
VAR
    lrDetectorTarget : LREAL;
    bDetectorSafe    : BOOL;
    bAllWarm         : BOOL;
END_VAR
M_StateMachine := FALSE;

lrDetectorTarget := nott_temps.out_lrLowestTemp + cfg.lrTemp_Det_OffSet;

bDetectorSafe :=
    nott_temps.out_bLowestTempValid
    AND nott_t_votes.vote_detector.stat.bValid
    AND (nott_t_votes.vote_detector.stat.lrTempK >= lrDetectorTarget);

bAllWarm :=
    nott_t_votes.vote_detector.stat.bValid
    AND nott_t_votes.vote_base_plate.stat.bValid
    AND nott_t_votes.vote_shield.stat.bValid
    AND nott_t_votes.vote_sidecar.stat.bValid
    AND nott_t_votes.vote_photonic_chip.stat.bValid
    AND (nott_t_votes.vote_detector.stat.lrTempK      >= cfg.lrTemp_Det)
    AND (nott_t_votes.vote_base_plate.stat.lrTempK    >= cfg.lrTemp_BasePlate)
    AND (nott_t_votes.vote_shield.stat.lrTempK        >= cfg.lrTemp_Shield)
    AND (nott_t_votes.vote_sidecar.stat.lrTempK       >= cfg.lrTemp_Sidecar)
    AND (nott_t_votes.vote_photonic_chip.stat.lrTempK >= cfg.lrTemp_PhotonicChip); 


CASE stat.nState OF

    E_NOTT_CRYO_WARMUP_STATE.NONE:
        stat.sState  := 'NONE';
        stat.sStatus := 'Undefined state';
        stat.nState  := E_NOTT_CRYO_WARMUP_STATE.OFF;


    E_NOTT_CRYO_WARMUP_STATE.OFF:

        stat.bActive := FALSE;
        stat.sState  := 'OFF';
        stat.sStatus := 'Warm-up OFF';

        out_bPermit_Evacuation_Stop := TRUE;
        out_bPermit_CoolDown        := TRUE;

        trig(CLK := in_bEnable);

        IF trig.Q
		   AND in_Cryo_Stat.bIsPVPRunning
		   AND in_Cryo_Stat.bIsTMPRunning THEN
            stat.bActive := TRUE;
            stat.nState := E_NOTT_CRYO_WARMUP_STATE.START_DETECTOR_PROTECTION;

            out_bPermit_Evacuation_Stop := FALSE;
            out_bPermit_CoolDown        := FALSE;
		ELSIF trig.Q THEN
			stat.sStatus := 'Warm-up start rejected: pumps not ready.';
        END_IF;


    E_NOTT_CRYO_WARMUP_STATE.START_DETECTOR_PROTECTION:

        out_bPermit_Evacuation_Stop := FALSE;
        out_bPermit_CoolDown        := FALSE;

        nott_heaters.h_detector.M_SetEnable();
        nott_heaters.h_detector_spare.M_SetEnable();

        nott_t_ctrls.tc_detector.M_SetEnable();
        nott_t_ctrls.tc_detector_spare.M_SetEnable();

        nott_t_ctrls.tc_detector.M_Set_SetPoint(
            m_eSetpointType    := E_METIS_CTRL_SETPOINT_SWITCH.FIXED,
            m_lrFixedSetpoint  := nott_temps.out_lrLowestTemp,
            m_lrSetpointOffset := cfg.lrTemp_Det_OffSet,
            m_pSetpointTemp    := nott_temps.M_SetTemperatureSensor(0)
        );

        nott_t_ctrls.tc_detector_spare.M_Set_SetPoint(
            m_eSetpointType    := E_METIS_CTRL_SETPOINT_SWITCH.FIXED,
            m_lrFixedSetpoint  := nott_temps.out_lrLowestTemp,
            m_lrSetpointOffset := cfg.lrTemp_Det_OffSet,
            m_pSetpointTemp    := nott_temps.M_SetTemperatureSensor(0)
        );

        stat.sState  := 'Detector protection';
        stat.sStatus := 'Waiting until detector is safely above lowest cryostat temperature';

        stat.nState := E_NOTT_CRYO_WARMUP_STATE.WAIT_DETECTOR_SAFE;


    E_NOTT_CRYO_WARMUP_STATE.WAIT_DETECTOR_SAFE:

        out_bPermit_Evacuation_Stop := FALSE;
        out_bPermit_CoolDown        := FALSE;

        // Keep detector protection active while waiting
        nott_t_ctrls.tc_detector.M_Set_SetPoint(
            m_eSetpointType    := E_METIS_CTRL_SETPOINT_SWITCH.FIXED,
            m_lrFixedSetpoint  := nott_temps.out_lrLowestTemp,
            m_lrSetpointOffset := cfg.lrTemp_Det_OffSet,
            m_pSetpointTemp    := nott_temps.M_SetTemperatureSensor(0)
        );

        nott_t_ctrls.tc_detector_spare.M_Set_SetPoint(
            m_eSetpointType    := E_METIS_CTRL_SETPOINT_SWITCH.FIXED,
            m_lrFixedSetpoint  := nott_temps.out_lrLowestTemp,
            m_lrSetpointOffset := cfg.lrTemp_Det_OffSet,
            m_pSetpointTemp    := nott_temps.M_SetTemperatureSensor(0)
        );

        IF NOT in_bEnable THEN
            stat.nState := E_NOTT_CRYO_WARMUP_STATE.STOP_WARMUP;
        ELSIF bDetectorSafe THEN
            stat.nState := E_NOTT_CRYO_WARMUP_STATE.START_WARMUP;
        ELSE
            stat.sStatus := 'Detector protection active...';
        END_IF;


    E_NOTT_CRYO_WARMUP_STATE.START_WARMUP:

        out_bPermit_Evacuation_Stop := FALSE;
        out_bPermit_CoolDown        := FALSE;

        // Enable remaining heaters
        nott_heaters.h_sidecar.M_SetEnable();
        nott_heaters.h_photonic_chip.M_SetEnable();
        nott_heaters.h_base_plate.M_SetEnable();
        nott_heaters.h_shield.M_SetEnable();

